(* Logix 5000 project; controller CarbonScout_MK6 vendor 1 type 14 code 154 rev 32.11; software revision 32.00; part 6 of 17 *)
(* tags used below, declared in another part *)
   Inp_OvrdCmd : DINT;   // Override Mode Command: 0=None, 1=Close, 2=Open
   Cfg_FailOpen : BOOL;   // 1=Fail Open (energize to close), 0=Fail Closed (energize to open)
   Cfg_PCmdClear : ALIAS FOR Mode.Cfg_PCmdClear;
   PSet_Owner : DINT;   // Program Owner Request ID (non-zero) or Release (zero)
   PCmd_Open : BOOL;   // Program Command to Open Valve
   PCmd_Close : BOOL;   // Program Command to Close Valve
   PCmd_Reset : BOOL;   // Program Command to Reset all Alarms requiring Reset
   OCmd_Open : BOOL;   // Operator Command to Open Valve
   OCmd_Close : BOOL;   // Operator Command to Close Valve
   OCmd_Bypass : BOOL;   // Operator Command to Bypass all Bypassable Interlocks and Permissives
   OCmd_Check : BOOL;   // Operator Command to Check (not bypass) all Interlocks and Permissives
   MCmd_Disable : BOOL;   // Maintenance Command to Disable Valve
   MCmd_Enable : BOOL;   // Maintenance Command to Enable (allow to energize) Valve
   OCmd_Reset : BOOL;   // Operator Command to Reset all Alarms requiring Reset
   OCmd_ResetAckAll : BOOL;   // Operator Command to Reset all Alarms and latched Shed conditions
   Out : BOOL;   // 1=Energize Valve Solenoid
   SrcQ_IO : DINT;   // Source and Quality of primary I/O (enumeration)
   SrcQ : DINT;   // Source and Quality of primary Val/Sts (enumeration)
   Val_Cmd : DINT;   // Device Command 0=None, 1=Close, 2=Open
   Val_Fdbk : DINT;   // Device Feedback 0=Moving, 1=Closed, 2=Opened, 3=Limit Switch Failure
   Val_Sts : DINT;   // Device Confirmed Sts 0=? 1=Closed 2=Open 5=Closing, 6=Opening, 33=Disabled
   Val_Fault : DINT;   // Device Fault Status 0=None, 16=Transit Stall, 17 = Full Stall, 32=I/O Fault, 34=Config Error
   Val_Mode : ALIAS FOR Mode.Val;
   Val_Owner : DINT;   // Current Object Owner ID (0=not owned)
   Val_Notify : DINT;   // Current Alarm Level and Acknowledgement (enumeration)
   Nrdy_Fail : BOOL;   // 1=Device Not Ready: Device Failure (Shed Requires Reset)
   Nrdy_IOFault : BOOL;   // 1=Device Not Ready: I/O Fault (Shed Requires Reset)
   Sts_MaintByp : BOOL;   // 1=A Maintenance Bypass is Active, display icon
   Sts_AlmInh : BOOL;   // 1=An Alarm is Shelved, Disabled or Suppressed, display icon
   Sts_Maint : ALIAS FOR Mode.Sts_Maint;
   Sts_Oper : ALIAS FOR Mode.Sts_Oper;
   Sts_NoMode : ALIAS FOR Mode.Sts_NoMode;
   Sts_IOFault : ALIAS FOR IOFault.Inp;   // I/O Comm Fault Status (0=OK, 1=Bad)
   Rdy_Disable : BOOL;   // 1=Ready to receive MCmd_Disable (enables HMI button)
   Rdy_Enable : BOOL;   // 1=Ready to receive MCmd_Enable (enables HMI button)
   Rdy_Reset : BOOL;   // 1=Ready to receive OCmd_Reset (enables HMI button)
   Rdy_ResetAckAll : BOOL;   // 1=At least one Alarm or latched Shed condition requires Reset or Ack
   P_ValveSO : BOOL;   // Unique Parameter Name for auto - discovery
   Mode : P_Mode;   // Valve Mode Selection
   IOFault : P_Alarm;   // I/O Fault Alarm
   IntlkTrip : P_Alarm;   // Interlock Trip Alarm
   TransitStall : P_Alarm;   // Valve Transit Stall (moved but did not reach target) Alarm
   FullStall : P_Alarm;   // Valve Full Stall (did not move) Alarm
   Wrk_Open : BOOL;   // 1=Requested to OPEN Valve, 0=Requested to CLOSE Valve
   Wrk_SimOpenT : TIMER;   // Simulation Delay until Opened
   Wrk_SimCloseT : TIMER;   // Simulation Delay until Closed
   Wrk_Notify : DINT;   // Buffer for building Val_Notify
   Wrk_TransitStallT : TIMER;   // Timer for Transit Stall Check
   Wrk_FullStallT : TIMER;   // Timer for Full Stall Check
   Wrk_SimOpenLS : BOOL;   // Simulated valve Open Limit Switch
   Wrk_SimClosedLS : BOOL;   // Simulated valve Closed Limit Switch
   test : DINT;
(* P_ValveSO, continued *)

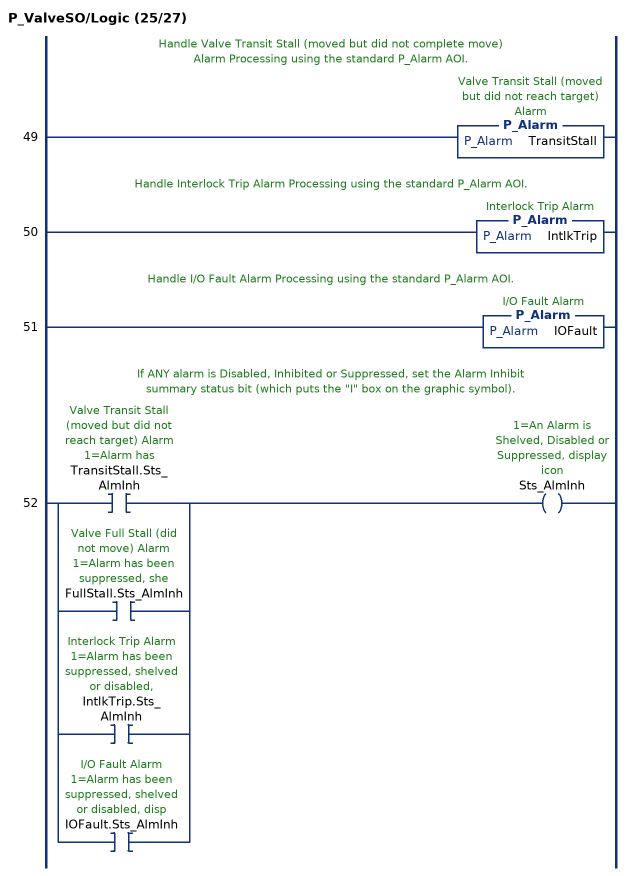
   // Handle Valve Transit Stall (moved but did not complete move)
   // Alarm Processing using the standard P_Alarm AOI.
   49: P_Alarm(TransitStall);
   // Handle Interlock Trip Alarm Processing using the standard P_Alarm AOI.
   50: P_Alarm(IntlkTrip);
   // Handle I/O Fault Alarm Processing using the standard P_Alarm AOI.
   51: P_Alarm(IOFault);
   // If ANY alarm is Disabled, Inhibited or Suppressed, set the Alarm Inhibit
   // summary status bit (which puts the "I" box on the graphic symbol).
   52: [XIC(TransitStall.Sts_AlmInh) ,XIC(FullStall.Sts_AlmInh) ,XIC(IntlkTrip.Sts_AlmInh) ,XIC(IOFault.Sts_AlmInh) ]OTE(Sts_AlmInh);
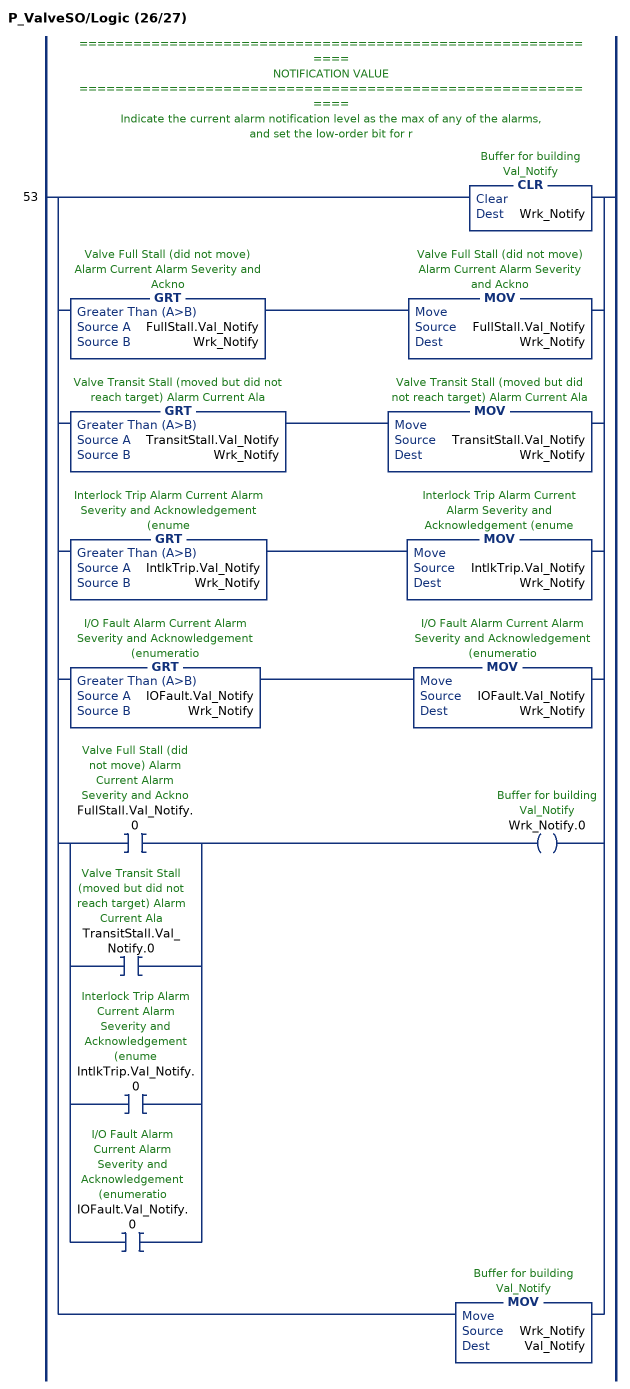
   // ============================================================
   // NOTIFICATION VALUE
   // ============================================================
   // Indicate the current alarm notification level as the max of any of the alarms,
   // and set the low-order bit for r
   53: [CLR(Wrk_Notify) ,GRT(FullStall.Val_Notify,Wrk_Notify) MOV(FullStall.Val_Notify,Wrk_Notify) ,GRT(TransitStall.Val_Notify,Wrk_Notify) MOV(TransitStall.Val_Notify,Wrk_Notify) ,GRT(IntlkTrip.Val_Notify,Wrk_Notify) MOV(IntlkTrip.Val_Notify,Wrk_Notify) ,GRT(IOFault.Val_Notify,Wrk_Notify) MOV(IOFault.Val_Notify,Wrk_Notify) ,[XIC(FullStall.Val_Notify.0) ,XIC(TransitStall.Val_Notify.0) ,XIC(IntlkTrip.Val_Notify.0) ,XIC(IOFault.Val_Notify.0) ] OTE(Wrk_Notify.0) ,MOV(Wrk_Notify,Val_Notify) ];
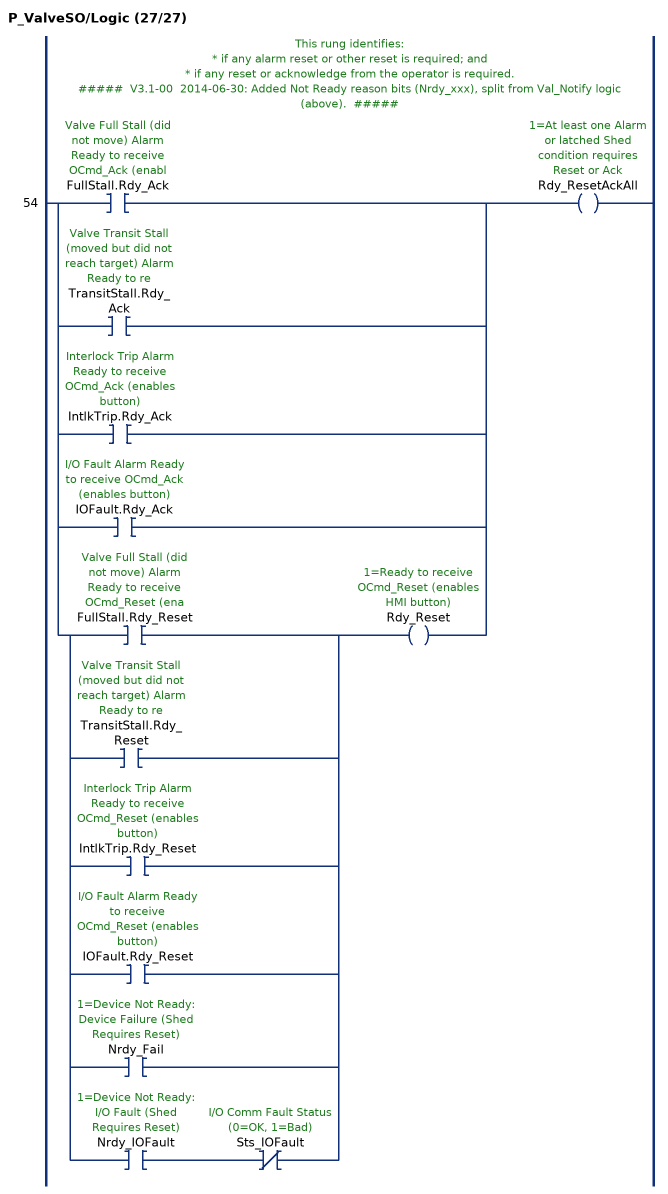
   // This rung identifies:
   // * if any alarm reset or other reset is required; and
   // * if any reset or acknowledge from the operator is required.
   // #####  V3.1-00  2014-06-30: Added Not Ready reason bits (Nrdy_xxx), split from Val_Notify logic (above).  #####
   54: [[XIC(FullStall.Rdy_Ack) ,XIC(TransitStall.Rdy_Ack) ,XIC(IntlkTrip.Rdy_Ack) ,XIC(IOFault.Rdy_Ack) ] ,[XIC(FullStall.Rdy_Reset) ,XIC(TransitStall.Rdy_Reset) ,XIC(IntlkTrip.Rdy_Reset) ,XIC(IOFault.Rdy_Reset) ,XIC(Nrdy_Fail) ,XIC(Nrdy_IOFault) XIO(Sts_IOFault) ] OTE(Rdy_Reset) ]OTE(Rdy_ResetAckAll);
END_ROUTINE

ROUTINE Prescan   (* ladder *)
// Clear Ownership, set to De-Energized state, clear "lurking" Commands
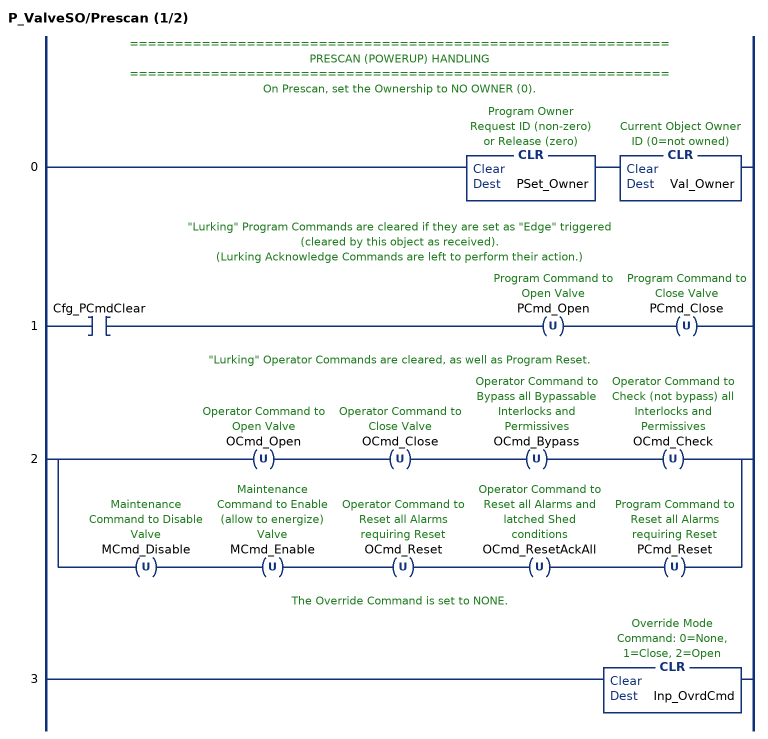
   // ============================================================
   // PRESCAN (POWERUP) HANDLING
   // ============================================================
   // On Prescan, set the Ownership to NO OWNER (0).
   0: CLR(PSet_Owner)CLR(Val_Owner);
   // "Lurking" Program Commands are cleared if they are set as "Edge" triggered
   // (cleared by this object as received).
   // (Lurking Acknowledge Commands are left to perform their action.)
   1: XIC(Cfg_PCmdClear)OTU(PCmd_Open)OTU(PCmd_Close);
   // "Lurking" Operator Commands are cleared, as well as Program Reset.
   2: [OTU(OCmd_Open) OTU(OCmd_Close) OTU(OCmd_Bypass) OTU(OCmd_Check) ,OTU(MCmd_Disable) OTU(MCmd_Enable) OTU(OCmd_Reset) OTU(OCmd_ResetAckAll) OTU(PCmd_Reset) ];
   // The Override Command is set to NONE.
   3: CLR(Inp_OvrdCmd);
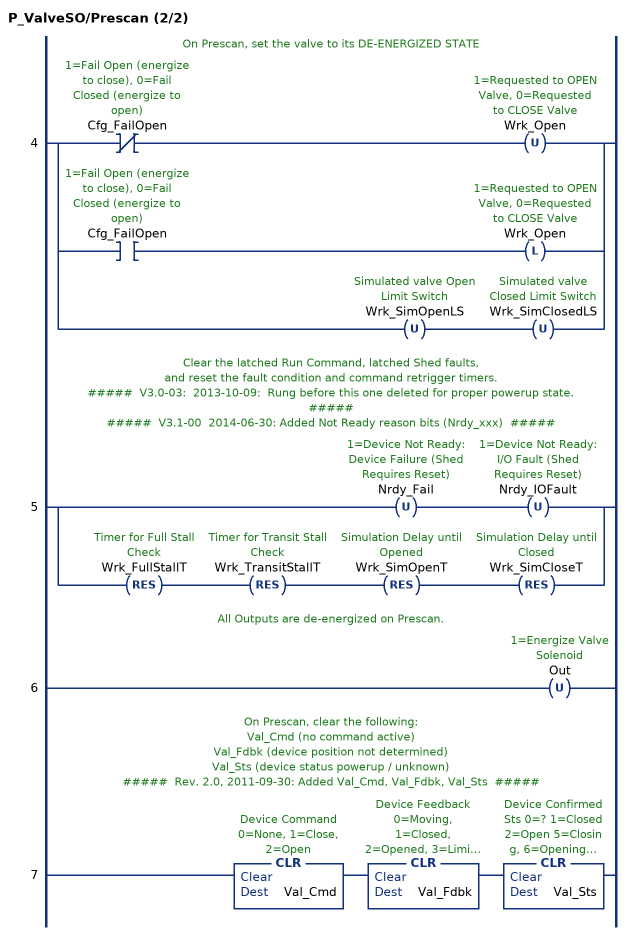
   // On Prescan, set the valve to its DE-ENERGIZED STATE
   4: [XIO(Cfg_FailOpen) OTU(Wrk_Open) ,XIC(Cfg_FailOpen) OTL(Wrk_Open) ,OTU(Wrk_SimOpenLS) OTU(Wrk_SimClosedLS) ];
   // Clear the latched Run Command, latched Shed faults,
   // and reset the fault condition and command retrigger timers.
   // #####  V3.0-03:  2013-10-09:  Rung before this one deleted for proper powerup state.  #####
   // #####  V3.1-00  2014-06-30: Added Not Ready reason bits (Nrdy_xxx)  #####
   5: [OTU(Nrdy_Fail) OTU(Nrdy_IOFault) ,RES(Wrk_FullStallT) RES(Wrk_TransitStallT) RES(Wrk_SimOpenT) RES(Wrk_SimCloseT) ];
   // All Outputs are de-energized on Prescan.
   6: OTU(Out);
   // On Prescan, clear the following:
   // Val_Cmd (no command active)
   // Val_Fdbk (device position not determined)
   // Val_Sts (device status powerup / unknown)
   // #####  Rev. 2.0, 2011-09-30: Added Val_Cmd, Val_Fdbk, Val_Sts  #####
   7: CLR(Val_Cmd)CLR(Val_Fdbk)CLR(Val_Sts);
END_ROUTINE
END_ADD_ON_INSTRUCTION

ADD_ON_INSTRUCTION TimerCompare   (* revision 1.0, ExecutePrescan *)
VAR_INPUT
   In_PresetTime1 : DINT; {required}
   In_PresetTime1_Multiplier : DINT; {required}
   In_PresetTime2 : DINT; {required}
   In_PresetTime2_Multiplier : DINT; {required}
   In_Time : DINT; {required}
END_VAR
VAR_OUTPUT
   Out_DN : BOOL;
END_VAR
VAR_INPUT
   In_ActiveStep : DINT; {required}
END_VAR
VAR
   Local_Time1 : DINT; {access None}
   Local_Time2 : DINT; {access None}
   Local_Time3 : DINT; {access None}
   LocalTimerDB : TIMER; {access None}
   LocalActiveStep : DINT; {access None}
END_VAR

ROUTINE Logic   (* ladder *)
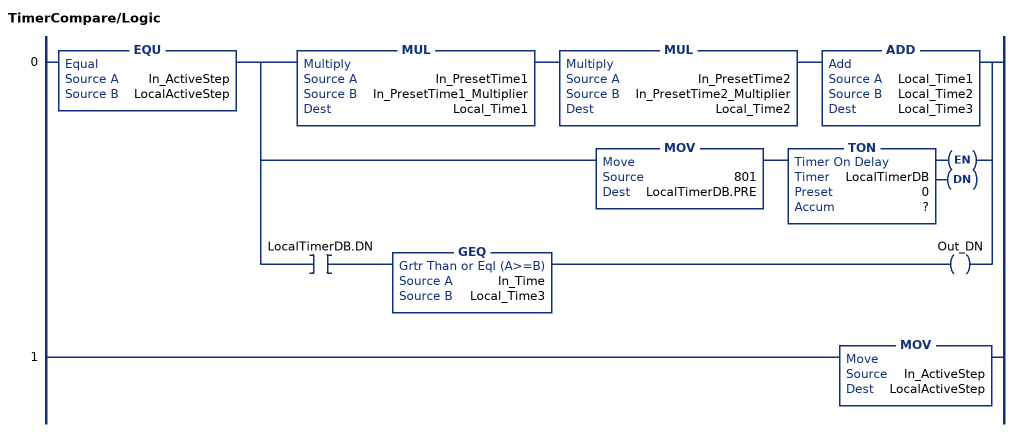
   0: EQU(In_ActiveStep,LocalActiveStep)[MUL(In_PresetTime1,In_PresetTime1_Multiplier,Local_Time1) MUL(In_PresetTime2,In_PresetTime2_Multiplier,Local_Time2) ADD(Local_Time1,Local_Time2,Local_Time3) ,MOV(801,LocalTimerDB.PRE) TON(LocalTimerDB,?,?) ,XIC(LocalTimerDB.DN) GEQ(In_Time,Local_Time3) OTE(Out_DN) ];
   1: MOV(In_ActiveStep,LocalActiveStep);
END_ROUTINE

ROUTINE Prescan   (* ladder *)
// Prescan
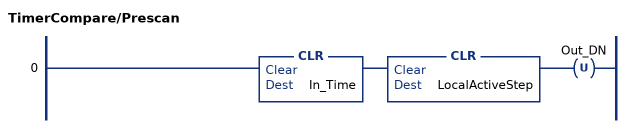
   0: CLR(In_Time)CLR(LocalActiveStep)OTU(Out_DN);
END_ROUTINE
END_ADD_ON_INSTRUCTION

ADD_ON_INSTRUCTION TimeRemainingCal   (* revision 1.0 *)
VAR_INPUT
   In_PresetTime : DINT; {visible}   // sec
END_VAR
VAR_OUTPUT
   RemainingHr : DINT; {required}
   RemainingMin : DINT; {required}
   RemainingSec : DINT; {required}
END_VAR
VAR_INPUT
   In_Time : DINT; {required}   // sec
END_VAR
VAR
   Local_Remaining : DINT; {access None}
   Local_RemainingMin : DINT; {access None}
   Local_Remainingsec : DINT; {access None}
END_VAR

ROUTINE Logic   (* ladder *)
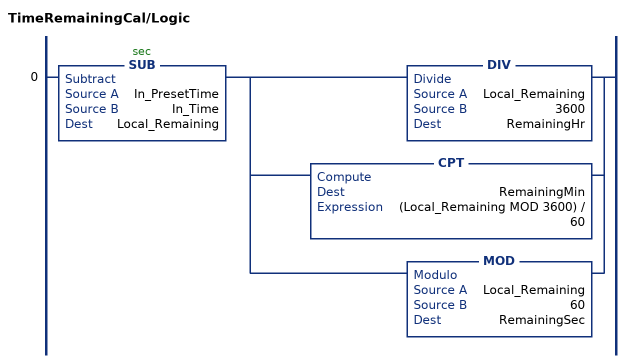
   0: SUB(In_PresetTime,In_Time,Local_Remaining)[DIV(Local_Remaining,3600,RemainingHr) ,CPT(RemainingMin,(Local_Remaining MOD 3600) / 60) ,MOD(Local_Remaining,60,RemainingSec) ];
END_ROUTINE
END_ADD_ON_INSTRUCTION

VAR_GLOBAL   (* controller tags *)
   a_Software_Version : STRING := '2.0.0';   // This must be updated and have a corrosponding change log and compadibility doc
   AI_AIT_01 : P_AIn := (Inp_PV := 9.085448, Inp_HiHiGate := 1, Inp_HiGate := 1, Inp_LoGate := 1, Inp_LoLoGate := 1, Inp_FailGate := 1, Cfg_SetTrack := 1, Cfg_PCmdClear := 1, Cfg_HiHiAckReqd := 1, Cfg_HiAckReqd := 1, Cfg_LoAckReqd := 1, Cfg_LoLoAckReqd := 1, Cfg_FailAckReqd := 1, Cfg_HiHiSeverity := 750, Cfg_HiSeverity := 500, Cfg_LoSeverity := 500, Cfg_LoLoSeverity := 750, Cfg_FailSeverity := 1000, Cfg_InpRawMax := 14.0, Cfg_PVEUMax := 14.0, Cfg_HiHiDB := 1.0, Cfg_HiDB := 1.0, Cfg_LoDB := 1.0, Cfg_LoLoDB := 1.0, Cfg_FailHiLim := 103.958336, Cfg_FailLoLim := -2.0833333, Cfg_FailDB := 0.41666666, Cfg_FailGateDly := 10, PSet_HiHiLim := 1.5e+38, PSet_HiLim := 1.5e+38, PSet_LoLim := -1.5e+38, PSet_LoLoLim := -1.5e+38, MSet_SubstPV := 9.085448, OSet_HiHiLim := 1.5e+38, OSet_HiLim := 1.5e+38, OSet_LoLim := -1.5e+38, OSet_LoLoLim := -1.5e+38, Set_SimPV := 9.085448, Val := 9.085448, Val_InpPV := 9.085448, Val_PVMinCapt := 9.085448, Val_PVMaxCapt := 9.085448, Val_PVEUMax := 14.0, SrcQ_IO := 1, SrcQ := 1, Val_Mode := 9, Val_HiHiLim := 1.5e+38, Val_HiLim := 1.5e+38, Val_LoLim := -1.5e+38, Val_LoLoLim := -1.5e+38, Sts_InpPV := 1, Sts_Oper := 1, Sts_HiHiGate := 1, Ack_HiHi := 1, Sts_HiGate := 1, Ack_Hi := 1, Sts_LoGate := 1, Ack_Lo := 1, Sts_LoLoGate := 1, Ack_LoLo := 1,
        Sts_FailGate := 1, Ack_Fail := 1, Rdy_OSet := 1);   // pH
   AI_AIT_02 : P_AIn := (Inp_PV := 6.017242, Inp_HiHiGate := 1, Inp_HiGate := 1, Inp_LoGate := 1, Inp_LoLoGate := 1, Inp_FailGate := 1, Cfg_SetTrack := 1, Cfg_PCmdClear := 1, Cfg_HiHiAckReqd := 1, Cfg_HiAckReqd := 1, Cfg_LoAckReqd := 1, Cfg_LoLoAckReqd := 1, Cfg_FailAckReqd := 1, Cfg_HiHiSeverity := 750, Cfg_HiSeverity := 500, Cfg_LoSeverity := 500, Cfg_LoLoSeverity := 750, Cfg_FailSeverity := 1000, Cfg_InpRawMax := 50.0, Cfg_PVEUMax := 50.0, Cfg_HiHiDB := 1.0, Cfg_HiDB := 1.0, Cfg_LoDB := 1.0, Cfg_LoLoDB := 1.0, Cfg_FailHiLim := 103.958336, Cfg_FailLoLim := -2.0833333, Cfg_FailDB := 0.41666666, Cfg_FailGateDly := 5, PSet_HiHiLim := 15000.0, PSet_HiLim := 15000.0, PSet_LoLim := -15000.0, PSet_LoLoLim := 15000.0, MSet_SubstPV := 39.0, OSet_HiHiLim := 15000.0, OSet_HiLim := 15000.0, OSet_LoLim := -15000.0, OSet_LoLoLim := 15000.0, Set_SimPV := 6.017242, Val := 39.0, Val_InpPV := 6.017242, Val_PVMinCapt := 39.0, Val_PVMaxCapt := 39.0, Val_PVEUMax := 50.0, SrcQ_IO := 1, SrcQ := 18, Val_Fault := 24, Val_Mode := 2, Val_HiHiLim := 15000.0, Val_HiLim := 15000.0, Val_LoLim := -15000.0, Val_LoLoLim := 15000.0, Sts_SubstPV := 1, Sts_MaintByp := 1, Sts_Maint := 1, Sts_HiHiGate := 1, Ack_HiHi := 1, Sts_HiGate := 1, Ack_Hi := 1, Sts_LoGate := 1, Ack_Lo := 1,
        Sts_LoLoCmp := 1, Sts_LoLoGate := 1, Sts_LoLo := 1, Ack_LoLo := 1, Sts_FailGate := 1, Ack_Fail := 1, Rdy_InpPV := 1, Rdy_OSet := 1);   // DO
   AI_AIT_03 : P_AIn := (Inp_HiHiGate := 1, Inp_HiGate := 1, Inp_LoGate := 1, Inp_LoLoGate := 1, Inp_FailGate := 1, Cfg_SetTrack := 1, Cfg_PCmdClear := 1, Cfg_HiHiAckReqd := 1, Cfg_HiAckReqd := 1, Cfg_LoAckReqd := 1, Cfg_LoLoAckReqd := 1, Cfg_FailAckReqd := 1, Cfg_HiHiSeverity := 750, Cfg_HiSeverity := 500, Cfg_LoSeverity := 500, Cfg_LoLoSeverity := 750, Cfg_FailSeverity := 1000, Cfg_InpRawMax := 100.0, Cfg_PVEUMax := 100.0, Cfg_HiHiDB := 1.0, Cfg_HiDB := 1.0, Cfg_LoDB := 1.0, Cfg_LoLoDB := 1.0, Cfg_FailHiLim := 103.958336, Cfg_FailLoLim := -2.0833333, Cfg_FailDB := 0.41666666, PSet_HiHiLim := 1.5e+38, PSet_HiLim := 1.5e+38, PSet_LoLim := -1.5e+38, PSet_LoLoLim := -1.5e+38, OSet_HiHiLim := 1.5e+38, OSet_HiLim := 1.5e+38, OSet_LoLim := -1.5e+38, OSet_LoLoLim := -1.5e+38, Val_PVMinCapt := 1.5e+38, Val_PVMaxCapt := -1.5e+38, Val_PVEUMax := 100.0, Val_HiHiLim := 1.5e+38, Val_HiLim := 1.5e+38, Val_LoLim := -1.5e+38, Val_LoLoLim := -1.5e+38, Sts_InpPV := 1, Sts_Oper := 1, Ack_HiHi := 1, Ack_Hi := 1, Ack_Lo := 1, Ack_LoLo := 1, Ack_Fail := 1);
   AI_Booster : P_AIn := (Inp_PV := 18408.0, Inp_HiHiGate := 1, Inp_HiGate := 1, Inp_LoGate := 1, Inp_LoLoGate := 1, Inp_FailGate := 1, Cfg_SetTrack := 1, Cfg_PCmdClear := 1, Cfg_HiHiAckReqd := 1, Cfg_HiAckReqd := 1, Cfg_LoAckReqd := 1, Cfg_LoLoAckReqd := 1, Cfg_FailAckReqd := 1, Cfg_HiHiSeverity := 750, Cfg_HiSeverity := 500, Cfg_LoSeverity := 500, Cfg_LoLoSeverity := 750, Cfg_FailSeverity := 1000, Cfg_InpRawMin := 4000.0, Cfg_InpRawMax := 20000.0, Cfg_PVEUMax := 100.0, Cfg_HiHiDB := 1.0, Cfg_HiDB := 1.0, Cfg_LoDB := 1.0, Cfg_LoOnDly := 1, Cfg_LoLoDB := 1.0, Cfg_LoLoOnDly := 1, Cfg_FailHiLim := 103.958336, Cfg_FailLoLim := -2.0833333, Cfg_FailDB := 0.41666666, PSet_HiHiLim := 95.0, PSet_HiLim := 80.0, PSet_LoLim := 25.0, PSet_LoLoLim := 10.0, MSet_SubstPV := 89.91875, OSet_HiHiLim := 95.0, OSet_HiLim := 80.0, OSet_LoLim := 25.0, OSet_LoLoLim := 10.0, Set_SimPV := 89.91875, Val := 89.91875, Val_InpPV := 89.91875, Val_PVMinCapt := 85.05625, Val_PVMaxCapt := 91.4, Val_PVEUMax := 100.0, SrcQ_IO := 1, SrcQ := 1, Val_Fault := 21, Val_Mode := 9, Val_HiHiLim := 95.0, Val_HiLim := 80.0, Val_LoLim := 25.0, Val_LoLoLim := 10.0, Sts_InpPV := 1, Sts_Oper := 1, Sts_HiHiGate := 1, Ack_HiHi := 1, Sts_HiCmp := 1, Sts_HiGate := 1, Sts_Hi := 1,
        Ack_Hi := 1, Sts_LoGate := 1, Ack_Lo := 1, Sts_LoLoGate := 1, Ack_LoLo := 1, Sts_FailGate := 1, Ack_Fail := 1, Rdy_OSet := 1);   // Booster Tank Level
   AI_FIT_01 : P_AIn := (Inp_PV := 4000.0, Inp_HiHiGate := 1, Inp_HiGate := 1, Inp_FailGate := 1, Cfg_SetTrack := 1, Cfg_PCmdClear := 1, Cfg_HasLoLoAlm := 1, Cfg_HasFailAlm := 1, Cfg_HiHiAckReqd := 1, Cfg_HiAckReqd := 1, Cfg_LoAckReqd := 1, Cfg_HiHiSeverity := 750, Cfg_HiSeverity := 500, Cfg_LoSeverity := 500, Cfg_LoLoSeverity := 750, Cfg_FailSeverity := 1000, Cfg_InpRawMin := 4000.0, Cfg_InpRawMax := 20000.0, Cfg_PVEUMax := 50.0, Cfg_HiHiDB := 1.0, Cfg_HiDB := 1.0, Cfg_LoDB := 1.0, Cfg_LoOnDly := 5, Cfg_LoGateDly := 5, Cfg_LoLoDB := 1.0, Cfg_LoLoOnDly := 5, Cfg_LoLoGateDly := 5, Cfg_FailHiLim := 55.0, Cfg_FailLoLim := -5.0, Cfg_FailDB := 0.41666666, PSet_HiHiLim := 1.5e+38, PSet_HiLim := 1.5e+38, PSet_LoLim := 0.5, PSet_LoLoLim := 0.3, OSet_HiHiLim := 1.5e+38, OSet_HiLim := 1.5e+38, OSet_LoLim := 0.5, OSet_LoLoLim := 0.3, Val_PVEUMax := 50.0, SrcQ_IO := 1, SrcQ := 1, Val_Mode := 9, Val_HiHiLim := 1.5e+38, Val_HiLim := 1.5e+38, Val_LoLim := 0.5, Val_LoLoLim := 0.3, Sts_InpPV := 1, Sts_Oper := 1, Sts_HiHiGate := 1, Ack_HiHi := 1, Sts_HiGate := 1, Ack_Hi := 1, Sts_LoCmp := 1, Ack_Lo := 1, Sts_LoLoCmp := 1, Ack_LoLo := 1, Sts_FailGate := 1, Ack_Fail := 1, Rdy_OSet := 1);   // Purge water flow
   AI_LIT_01 : P_AIn := (Inp_PV := 20489.0, Inp_HiHiGate := 1, Inp_HiGate := 1, Inp_LoGate := 1, Inp_LoLoGate := 1, Inp_FailGate := 1, Cfg_SetTrack := 1, Cfg_HasChanObj := 1, Cfg_PCmdClear := 1, Cfg_HiHiAckReqd := 1, Cfg_HiAckReqd := 1, Cfg_LoAckReqd := 1, Cfg_LoLoAckReqd := 1, Cfg_HiHiSeverity := 750, Cfg_HiSeverity := 500, Cfg_LoSeverity := 500, Cfg_LoLoSeverity := 750, Cfg_FailSeverity := 1000, Cfg_InpRawMin := 4000.0, Cfg_InpRawMax := 20000.0, Cfg_PVEUMin := 192.0, Cfg_PVEUMax := 1410.0, Cfg_FiltTC := 0.2, Cfg_HiHiDB := 1.0, Cfg_HiDB := 1.0, Cfg_LoDB := 1.0, Cfg_LoLoDB := 1.0, Cfg_FailHiLim := 1480.0, Cfg_FailLoLim := 180.0, Cfg_FailDB := 5.0, Cfg_FailGateDly := 10, PSet_HiHiLim := 1475.0, PSet_HiLim := 1.5e+38, PSet_LoLim := -1.5e+38, PSet_LoLoLim := 180.0, MSet_SubstPV := 1447.2251, OSet_HiHiLim := 1475.0, OSet_HiLim := 1.5e+38, OSet_LoLim := -1.5e+38, OSet_LoLoLim := 180.0, Set_SimPV := 1447.2251, Val := 1447.2251, Val_InpPV := 1447.2251, Val_PVMinCapt := 1447.2251, Val_PVMaxCapt := 1447.2251, Val_PVEUMin := 192.0, Val_PVEUMax := 1410.0, SrcQ_IO := 1, SrcQ := 1, Val_Mode := 9, Val_HiHiLim := 1475.0, Val_HiLim := 1.5e+38, Val_LoLim := -1.5e+38, Val_LoLoLim := 180.0, Sts_InpPV := 1, Sts_Oper := 1, Sts_HiHiGate := 1, Ack_HiHi := 1, Sts_HiGate := 1, Ack_Hi := 1,
        Sts_LoGate := 1, Ack_Lo := 1, Sts_LoLoGate := 1, Ack_LoLo := 1, Sts_FailGate := 1, Ack_Fail := 1, Rdy_OSet := 1);   // Carbon Scout Laser Level Transmitter
   AI_LIT_02 : P_AIn := (Inp_PV := 0.0015260963, Inp_HiHiGate := 1, Inp_HiGate := 1, Inp_LoGate := 1, Inp_LoLoGate := 1, Inp_FailGate := 1, Cfg_SetTrack := 1, Cfg_PCmdClear := 1, Cfg_HasFailAlm := 1, Cfg_HiHiAckReqd := 1, Cfg_HiAckReqd := 1, Cfg_LoAckReqd := 1, Cfg_LoLoAckReqd := 1, Cfg_HiHiSeverity := 750, Cfg_HiSeverity := 500, Cfg_LoSeverity := 500, Cfg_LoLoSeverity := 750, Cfg_FailSeverity := 1000, Cfg_InpRawMax := 20.0, Cfg_PVEUMax := 20.0, Cfg_HiHiDB := 1.0, Cfg_HiDB := 1.0, Cfg_LoDB := 1.0, Cfg_LoLoDB := 1.0, Cfg_FailHiLim := 25.0, Cfg_FailLoLim := -1.0, Cfg_FailDB := 0.5, Cfg_FailGateDly := 10, PSet_HiHiLim := 20.0, PSet_HiLim := 1.5e+38, PSet_LoLoLim := 3.8, MSet_SubstPV := 0.0015260963, OSet_HiHiLim := 20.0, OSet_HiLim := 1.5e+38, OSet_LoLoLim := 3.8, Set_SimPV := 0.0015260963, Val := 0.0015260963, Val_InpPV := 0.0015260963, Val_PVMinCapt := 0.0015260963, Val_PVMaxCapt := 0.0015260963, Val_PVEUMax := 20.0, SrcQ_IO := 1, SrcQ := 1, Val_Fault := 24, Val_Mode := 2, Val_HiHiLim := 20.0, Val_HiLim := 1.5e+38, Val_LoLoLim := 3.8, Sts_InpPV := 1, Sts_Maint := 1, Sts_HiHiGate := 1, Ack_HiHi := 1, Sts_HiGate := 1, Ack_Hi := 1, Sts_LoGate := 1, Ack_Lo := 1, Sts_LoLoCmp := 1, Sts_LoLoGate := 1, Sts_LoLo := 1, Ack_LoLo := 1,
        Sts_FailGate := 1, Ack_Fail := 1, Rdy_SubstPV := 1, Rdy_OSet := 1);   // Carbon Scout Cone Level Transmitter
   AI_PIT_01 : P_AIn := (Inp_PV := 12000.0, Inp_HiHiGate := 1, Inp_HiGate := 1, Inp_LoGate := 1, Inp_LoLoGate := 1, Inp_FailGate := 1, Cfg_SetTrack := 1, Cfg_PCmdClear := 1, Cfg_HasLoAlm := 1, Cfg_HasLoLoAlm := 1, Cfg_HasFailAlm := 1, Cfg_HiHiAckReqd := 1, Cfg_HiAckReqd := 1, Cfg_HiHiSeverity := 750, Cfg_HiSeverity := 500, Cfg_LoSeverity := 500, Cfg_LoLoSeverity := 750, Cfg_FailSeverity := 1000, Cfg_InpRawMin := 4000.0, Cfg_InpRawMax := 20000.0, Cfg_PVEUMax := 1000.0, Cfg_FiltTC := 1.0, Cfg_HiHiDB := 1.0, Cfg_HiDB := 1.0, Cfg_LoDB := 1.0, Cfg_LoOnDly := 5, Cfg_LoLoDB := 1.0, Cfg_LoLoOnDly := 60, Cfg_FailHiLim := 1100.0, Cfg_FailLoLim := -100.0, Cfg_FailDB := 0.41666666, Cfg_FailGateDly := 5, PSet_HiHiLim := 650.0, PSet_HiLim := 630.0, PSet_LoLim := 120.0, PSet_LoLoLim := 90.0, MSet_SubstPV := 500.0, OSet_HiHiLim := 650.0, OSet_HiLim := 630.0, OSet_LoLim := 120.0, OSet_LoLoLim := 90.0, Set_SimPV := 500.0, Val := 500.0, Val_InpPV := 500.0, Val_PVMinCapt := 500.0, Val_PVMaxCapt := 500.0, Val_PVEUMax := 1000.0, SrcQ_IO := 1, SrcQ := 1, Val_Mode := 9, Val_HiHiLim := 650.0, Val_HiLim := 630.0, Val_LoLim := 120.0, Val_LoLoLim := 90.0, Sts_InpPV := 1, Sts_Oper := 1, Sts_HiHiGate := 1, Ack_HiHi := 1, Sts_HiGate := 1, Ack_Hi := 1,
        Sts_LoGate := 1, Ack_Lo := 1, Sts_LoLoGate := 1, Ack_LoLo := 1, Sts_FailGate := 1, Ack_Fail := 1, Rdy_OSet := 1);   // Water supply pressure
   AI_TIT_01 : P_AIn := (Inp_HiHiGate := 1, Inp_HiGate := 1, Inp_LoGate := 1, Inp_LoLoGate := 1, Inp_FailGate := 1, Cfg_SetTrack := 1, Cfg_PCmdClear := 1, Cfg_HiHiAckReqd := 1, Cfg_HiAckReqd := 1, Cfg_LoAckReqd := 1, Cfg_LoLoAckReqd := 1, Cfg_FailAckReqd := 1, Cfg_HiHiSeverity := 750, Cfg_HiSeverity := 500, Cfg_LoSeverity := 500, Cfg_LoLoSeverity := 750, Cfg_FailSeverity := 1000, Cfg_InpRawMax := 50.0, Cfg_PVEUMax := 50.0, Cfg_HiHiDB := 1.0, Cfg_HiDB := 1.0, Cfg_LoDB := 1.0, Cfg_LoLoDB := 1.0, Cfg_FailHiLim := 103.958336, Cfg_FailLoLim := -2.0833333, Cfg_FailDB := 0.41666666, Cfg_FailGateDly := 5, PSet_HiHiLim := 1.5e+38, PSet_HiLim := 1.5e+38, PSet_LoLim := -1.5e+38, PSet_LoLoLim := -1.5e+38, OSet_HiHiLim := 1.5e+38, OSet_HiLim := 1.5e+38, OSet_LoLim := -1.5e+38, OSet_LoLoLim := -1.5e+38, Val_PVEUMax := 50.0, SrcQ_IO := 1, SrcQ := 1, Val_Mode := 9, Val_HiHiLim := 1.5e+38, Val_HiLim := 1.5e+38, Val_LoLim := -1.5e+38, Val_LoLoLim := -1.5e+38, Sts_InpPV := 1, Sts_Oper := 1, Sts_HiHiGate := 1, Ack_HiHi := 1, Sts_HiGate := 1, Ack_Hi := 1, Sts_LoGate := 1, Ack_Lo := 1, Sts_LoLoGate := 1, Ack_LoLo := 1, Sts_FailGate := 1, Ack_Fail := 1, Rdy_OSet := 1);   // Temperature
   AI_WIT_01 : P_AIn := (Inp_PV := -5.0, Inp_HiHiGate := 1, Inp_HiGate := 1, Inp_LoGate := 1, Inp_LoLoGate := 1, Inp_FailGate := 1, Cfg_SetTrack := 1, Cfg_PCmdClear := 1, Cfg_HasFailAlm := 1, Cfg_HiHiAckReqd := 1, Cfg_HiAckReqd := 1, Cfg_LoAckReqd := 1, Cfg_LoLoAckReqd := 1, Cfg_HiHiSeverity := 750, Cfg_HiSeverity := 500, Cfg_LoSeverity := 500, Cfg_LoLoSeverity := 750, Cfg_FailSeverity := 1000, Cfg_InpRawMin := 4000.0, Cfg_InpRawMax := 20000.0, Cfg_PVEUMin := 2.0, Cfg_PVEUMax := 52.0, Cfg_FiltTC := 1.0, Cfg_HiHiDB := 1.0, Cfg_HiDB := 1.0, Cfg_LoDB := 1.0, Cfg_LoLoDB := 1.0, Cfg_FailHiLim := 52.5, Cfg_FailLoLim := -5.0, Cfg_FailDB := 0.5, Cfg_FailGateDly := 5, PSet_HiHiLim := 1.5e+38, PSet_HiLim := 1.5e+38, PSet_LoLim := -1.5e+38, PSet_LoLoLim := -1.5e+38, MSet_SubstPV := -10.521875, OSet_HiHiLim := 1.5e+38, OSet_HiLim := 1.5e+38, OSet_LoLim := -1.5e+38, OSet_LoLoLim := -1.5e+38, Set_SimPV := -10.521875, PCmd_ClearCapt := 1, Val := -10.52187, Val_InpPV := -10.515625, Val_PVMinCapt := -10.52187, Val_PVMaxCapt := -10.51875, Val_PVEUMin := 2.0, Val_PVEUMax := 52.0, SrcQ_IO := 32, SrcQ := 19, Val_HiHiLim := 1.5e+38, Val_HiLim := 1.5e+38, Val_LoLim := -1.5e+38, Val_LoLoLim := -1.5e+38, Sts_PVBad := 1, Sts_AlmInh := 1, Sts_NoMode := 1, Ack_HiHi := 1, Ack_Hi := 1, Ack_Lo := 1,
        Ack_LoLo := 1, Ack_Fail := 1);   // Weight measure
   Client_to_Gekko : DINT[10] := ([0] := 64);
        [0].0   // Command Start Carbon Scout
        [0].1   // Command Pause Carbon Scout
        [0].15   // Take Tank Offline 16
        [0].16   // Take Tank Offline 1
        [0].17   // Take Tank Offline 2
        [0].18   // Take Tank Offline 3
        [0].19   // Take Tank Offline 4
        [0].2   // Command Shutdown Carbon Scout
        [0].20   // Take Tank Offline 5
        [0].21   // Take Tank Offline 6
        [0].22   // Take Tank Offline 7
        [0].23   // Take Tank Offline 8
        [0].24   // Take Tank Offline 9
        [0].25   // Take Tank Offline 10
        [0].26   // Take Tank Offline 11
        [0].27   // Take Tank Offline 12
        [0].28   // Take Tank Offline 13
        [0].29   // Take Tank Offline 14
        [0].3   // Command All Drives / Valves to Auto
        [0].30   // Take Tank Offline 15
        [0].4   // Command - Reset All Faults / Alarms
        [0].5   // Command Crash Stop Carbon Scout
        [0].6   // Indicate Newmont water supply is ok
        [0].7   // Tank HOld Request
        [0].8   // Enable Remote mode
        [0].9   // Remote Auto/Man Request 1 = Auto, 0 = Man
   CS_Alarms : P_Alarm[80] := ([0].Cfg_Exists := 1, [0].Cfg_AllowShelve := 1, [0].Cfg_AllowDisable := 1, [0].Cfg_PCmdClear := 1, [0].Cfg_Severity := 750, [0].Cfg_AlmMinOnT := 5, [0].Cfg_MaxShelfT := 480, [0].PCfg_AllowExist := 1, [0].Ack := 1, [0].Rdy_Shelve := 1, [0].Rdy_Disable := 1, [0].Rdy_Test := 1, [1].Cfg_Exists := 1, [1].Cfg_ResetReqd := 1, [1].Cfg_AllowShelve := 1, [1].Cfg_AllowDisable := 1, [1].Cfg_PCmdClear := 1, [1].Cfg_Severity := 750, [1].Cfg_AlmMinOnT := 5, [1].Cfg_MaxShelfT := 480, [1].PCfg_AllowExist := 1, [1].Ack := 1, [1].Rdy_Shelve := 1, [1].Rdy_Disable := 1, [1].Rdy_Test := 1, [2].Cfg_Exists := 1, [2].Cfg_AllowShelve := 1, [2].Cfg_AllowDisable := 1, [2].Cfg_PCmdClear := 1, [2].Cfg_Severity := 750, [2].Cfg_AlmMinOnT := 5, [2].Cfg_MaxShelfT := 480, [2].PCfg_AllowExist := 1, [2].Ack := 1, [2].Rdy_Shelve := 1, [2].Rdy_Disable := 1, [2].Rdy_Test := 1, [3].Cfg_Exists := 1, [3].Cfg_AllowShelve := 1, [3].Cfg_AllowDisable := 1, [3].Cfg_PCmdClear := 1, [3].Cfg_Severity := 750, [3].Cfg_AlmMinOnT := 5, [3].Cfg_MaxShelfT := 480, [3].PCfg_AllowExist := 1, [3].Ack := 1, [3].Rdy_Shelve := 1, [3].Rdy_Disable := 1, [3].Rdy_Test := 1, [4].Cfg_Exists := 1, [4].Cfg_AllowShelve := 1, [4].Cfg_AllowDisable := 1, [4].Cfg_PCmdClear := 1, [4].Cfg_Severity := 750, [4].Cfg_AlmMinOnT := 5, [4].Cfg_MaxShelfT := 480, [4].PCfg_AllowExist := 1, [4].Ack := 1, [4].Rdy_Shelve := 1, [4].Rdy_Disable := 1,
        [4].Rdy_Test := 1, [5].Cfg_Exists := 1, [5].Cfg_AllowShelve := 1, [5].Cfg_AllowDisable := 1, [5].Cfg_PCmdClear := 1, [5].Cfg_Severity := 750, [5].Cfg_AlmMinOnT := 5, [5].Cfg_MaxShelfT := 480, [5].PCfg_AllowExist := 1, [5].Ack := 1, [5].Rdy_Shelve := 1, [5].Rdy_Disable := 1, [5].Rdy_Test := 1, [6].Cfg_Exists := 1, [6].Cfg_AllowShelve := 1, [6].Cfg_AllowDisable := 1, [6].Cfg_PCmdClear := 1, [6].Cfg_Severity := 750, [6].Cfg_AlmMinOnT := 5, [6].Cfg_MaxShelfT := 480, [6].PCfg_AllowExist := 1, [6].Ack := 1, [6].Rdy_Shelve := 1, [6].Rdy_Disable := 1, [6].Rdy_Test := 1, [7].Cfg_Exists := 1, [7].Cfg_AllowShelve := 1, [7].Cfg_AllowDisable := 1, [7].Cfg_PCmdClear := 1, [7].Cfg_Severity := 750, [7].Cfg_AlmMinOnT := 5, [7].Cfg_MaxShelfT := 480, [7].PCfg_AllowExist := 1, [7].Ack := 1, [7].Rdy_Shelve := 1, [7].Rdy_Disable := 1, [7].Rdy_Test := 1, [8].Cfg_Exists := 1, [8].Cfg_AllowShelve := 1, [8].Cfg_AllowDisable := 1, [8].Cfg_PCmdClear := 1, [8].Cfg_Severity := 750, [8].Cfg_AlmMinOnT := 5, [8].Cfg_MaxShelfT := 480, [8].PCfg_AllowExist := 1, [8].Ack := 1, [8].Rdy_Shelve := 1, [8].Rdy_Disable := 1, [8].Rdy_Test := 1, [9].Cfg_Exists := 1, [9].Cfg_AllowShelve := 1, [9].Cfg_AllowDisable := 1, [9].Cfg_PCmdClear := 1, [9].Cfg_Severity := 750, [9].Cfg_AlmMinOnT := 5, [9].Cfg_MaxShelfT := 480, [9].PCfg_AllowExist := 1, [9].Ack := 1, [9].Rdy_Shelve := 1, [9].Rdy_Disable := 1,
        [9].Rdy_Test := 1, [10].Cfg_Exists := 1, [10].Cfg_AllowShelve := 1, [10].Cfg_AllowDisable := 1, [10].Cfg_PCmdClear := 1, [10].Cfg_Severity := 750, [10].Cfg_AlmMinOnT := 5, [10].Cfg_MaxShelfT := 480, [10].PCfg_AllowExist := 1, [10].Ack := 1, [10].Rdy_Shelve := 1, [10].Rdy_Disable := 1, [10].Rdy_Test := 1, [11].Cfg_Exists := 1, [11].Cfg_AllowShelve := 1, [11].Cfg_AllowDisable := 1, [11].Cfg_PCmdClear := 1, [11].Cfg_Severity := 750, [11].Cfg_AlmMinOnT := 5, [11].Cfg_MaxShelfT := 480, [11].PCfg_AllowExist := 1, [11].Ack := 1, [11].Rdy_Shelve := 1, [11].Rdy_Disable := 1, [11].Rdy_Test := 1, [12].Cfg_Exists := 1, [12].Cfg_AllowShelve := 1, [12].Cfg_AllowDisable := 1, [12].Cfg_PCmdClear := 1, [12].Cfg_Severity := 750, [12].Cfg_AlmMinOnT := 5, [12].Cfg_MaxShelfT := 480, [12].PCfg_AllowExist := 1, [12].Ack := 1, [12].Rdy_Shelve := 1, [12].Rdy_Disable := 1, [12].Rdy_Test := 1, [13].Cfg_Exists := 1, [13].Cfg_AllowShelve := 1, [13].Cfg_AllowDisable := 1, [13].Cfg_PCmdClear := 1, [13].Cfg_Severity := 750, [13].Cfg_AlmMinOnT := 5, [13].Cfg_MaxShelfT := 480, [13].PCfg_AllowExist := 1, [13].Ack := 1, [13].Rdy_Shelve := 1, [13].Rdy_Disable := 1, [13].Rdy_Test := 1, [14].Cfg_Exists := 1, [14].Cfg_ResetReqd := 1, [14].Cfg_AllowShelve := 1, [14].Cfg_AllowDisable := 1, [14].Cfg_PCmdClear := 1, [14].Cfg_Severity := 750, [14].Cfg_AlmMinOnT := 5, [14].Cfg_MaxShelfT := 480, [14].PCfg_AllowExist := 1, [14].Ack := 1, [14].Rdy_Shelve := 1,
        [14].Rdy_Disable := 1, [14].Rdy_Test := 1, [15].Cfg_Exists := 1, [15].Cfg_ResetReqd := 1, [15].Cfg_AllowShelve := 1, [15].Cfg_AllowDisable := 1, [15].Cfg_PCmdClear := 1, [15].Cfg_Severity := 750, [15].Cfg_AlmMinOnT := 5, [15].Cfg_MaxShelfT := 480, [15].PCfg_AllowExist := 1, [15].Ack := 1, [15].Rdy_Shelve := 1, [15].Rdy_Disable := 1, [15].Rdy_Test := 1, [16].Cfg_Exists := 1, [16].Cfg_ResetReqd := 1, [16].Cfg_AllowShelve := 1, [16].Cfg_AllowDisable := 1, [16].Cfg_PCmdClear := 1, [16].Cfg_Severity := 750, [16].Cfg_AlmMinOnT := 5, [16].Cfg_MaxShelfT := 480, [16].PCfg_AllowExist := 1, [16].Ack := 1, [16].Rdy_Shelve := 1, [16].Rdy_Disable := 1, [16].Rdy_Test := 1, [17].Cfg_Exists := 1, [17].Cfg_ResetReqd := 1, [17].Cfg_AllowShelve := 1, [17].Cfg_AllowDisable := 1, [17].Cfg_PCmdClear := 1, [17].Cfg_Severity := 750, [17].Cfg_AlmMinOnT := 5, [17].Cfg_MaxShelfT := 480, [17].PCfg_AllowExist := 1, [17].Ack := 1, [17].Rdy_Shelve := 1, [17].Rdy_Disable := 1, [17].Rdy_Test := 1, [18].Cfg_Exists := 1, [18].Cfg_ResetReqd := 1, [18].Cfg_AllowShelve := 1, [18].Cfg_AllowDisable := 1, [18].Cfg_PCmdClear := 1, [18].Cfg_Severity := 750, [18].Cfg_AlmMinOnT := 5, [18].Cfg_MaxShelfT := 480, [18].PCfg_AllowExist := 1, [18].Ack := 1, [18].Rdy_Shelve := 1, [18].Rdy_Disable := 1, [18].Rdy_Test := 1, [19].Cfg_Exists := 1, [19].Cfg_ResetReqd := 1, [19].Cfg_AllowShelve := 1, [19].Cfg_AllowDisable := 1, [19].Cfg_PCmdClear := 1, [19].Cfg_Severity := 750,
        [19].Cfg_AlmMinOnT := 5, [19].Cfg_MaxShelfT := 480, [19].PCfg_AllowExist := 1, [19].Ack := 1, [19].Rdy_Shelve := 1, [19].Rdy_Disable := 1, [19].Rdy_Test := 1, [20].Cfg_Exists := 1, [20].Cfg_ResetReqd := 1, [20].Cfg_AllowShelve := 1, [20].Cfg_AllowDisable := 1, [20].Cfg_PCmdClear := 1, [20].Cfg_Severity := 750, [20].Cfg_AlmMinOnT := 5, [20].Cfg_MaxShelfT := 480, [20].PCfg_AllowExist := 1, [20].Ack := 1, [20].Rdy_Shelve := 1, [20].Rdy_Disable := 1, [20].Rdy_Test := 1, [21].Cfg_Exists := 1, [21].Cfg_ResetReqd := 1, [21].Cfg_AllowShelve := 1, [21].Cfg_AllowDisable := 1, [21].Cfg_PCmdClear := 1, [21].Cfg_Severity := 750, [21].Cfg_AlmMinOnT := 5, [21].Cfg_MaxShelfT := 480, [21].PCfg_AllowExist := 1, [21].Ack := 1, [21].Rdy_Shelve := 1, [21].Rdy_Disable := 1, [21].Rdy_Test := 1, [22].Cfg_Exists := 1, [22].Cfg_ResetReqd := 1, [22].Cfg_AllowShelve := 1, [22].Cfg_AllowDisable := 1, [22].Cfg_PCmdClear := 1, [22].Cfg_Severity := 750, [22].Cfg_AlmMinOnT := 5, [22].Cfg_MaxShelfT := 480, [22].PCfg_AllowExist := 1, [22].Ack := 1, [22].Rdy_Shelve := 1, [22].Rdy_Disable := 1, [22].Rdy_Test := 1, [23].Cfg_Exists := 1, [23].Cfg_ResetReqd := 1, [23].Cfg_AllowShelve := 1, [23].Cfg_AllowDisable := 1, [23].Cfg_PCmdClear := 1, [23].Cfg_Severity := 750, [23].Cfg_AlmMinOnT := 5, [23].Cfg_MaxShelfT := 480, [23].PCfg_AllowExist := 1, [23].Ack := 1, [23].Rdy_Shelve := 1, [23].Rdy_Disable := 1, [23].Rdy_Test := 1, [24].Cfg_Exists := 1,
        [24].Cfg_ResetReqd := 1, [24].Cfg_AllowShelve := 1, [24].Cfg_AllowDisable := 1, [24].Cfg_PCmdClear := 1, [24].Cfg_Severity := 750, [24].Cfg_AlmMinOnT := 5, [24].Cfg_MaxShelfT := 480, [24].PCfg_AllowExist := 1, [24].Ack := 1, [24].Rdy_Shelve := 1, [24].Rdy_Disable := 1, [24].Rdy_Test := 1, [25].Cfg_Exists := 1, [25].Cfg_AllowShelve := 1, [25].Cfg_AllowDisable := 1, [25].Cfg_PCmdClear := 1, [25].Cfg_Severity := 750, [25].Cfg_AlmMinOnT := 5, [25].Cfg_MaxShelfT := 480, [25].PCfg_AllowExist := 1, [25].Ack := 1, [25].Rdy_Shelve := 1, [25].Rdy_Disable := 1, [25].Rdy_Test := 1, [26].Cfg_Exists := 1, [26].Cfg_AllowShelve := 1, [26].Cfg_AllowDisable := 1, [26].Cfg_PCmdClear := 1, [26].Cfg_Severity := 750, [26].Cfg_AlmMinOnT := 5, [26].Cfg_MaxShelfT := 480, [26].PCfg_AllowExist := 1, [26].Ack := 1, [26].Rdy_Shelve := 1, [26].Rdy_Disable := 1, [26].Rdy_Test := 1, [27].Cfg_Exists := 1, [27].Cfg_AllowShelve := 1, [27].Cfg_AllowDisable := 1, [27].Cfg_PCmdClear := 1, [27].Cfg_Severity := 750, [27].Cfg_AlmMinOnT := 5, [27].Cfg_MaxShelfT := 480, [27].PCfg_AllowExist := 1, [27].Ack := 1, [27].Rdy_Shelve := 1, [27].Rdy_Disable := 1, [27].Rdy_Test := 1, [28].Cfg_Exists := 1, [28].Cfg_AllowShelve := 1, [28].Cfg_AllowDisable := 1, [28].Cfg_PCmdClear := 1, [28].Cfg_Severity := 750, [28].Cfg_AlmMinOnT := 5, [28].Cfg_MaxShelfT := 480, [28].PCfg_AllowExist := 1, [28].Ack := 1, [28].Rdy_Shelve := 1, [28].Rdy_Disable := 1, [28].Rdy_Test := 1,
        [29].Cfg_Exists := 1, [29].Cfg_AllowShelve := 1, [29].Cfg_AllowDisable := 1, [29].Cfg_PCmdClear := 1, [29].Cfg_Severity := 750, [29].Cfg_AlmMinOnT := 5, [29].Cfg_MaxShelfT := 480, [29].PCfg_AllowExist := 1, [29].Ack := 1, [29].Rdy_Shelve := 1, [29].Rdy_Disable := 1, [29].Rdy_Test := 1, [30].Cfg_Exists := 1, [30].Cfg_AllowShelve := 1, [30].Cfg_AllowDisable := 1, [30].Cfg_PCmdClear := 1, [30].Cfg_Severity := 750, [30].Cfg_AlmMinOnT := 5, [30].Cfg_MaxShelfT := 480, [30].PCfg_AllowExist := 1, [30].Ack := 1, [30].Rdy_Shelve := 1, [30].Rdy_Disable := 1, [30].Rdy_Test := 1, [31].Cfg_Exists := 1, [31].Cfg_AllowShelve := 1, [31].Cfg_AllowDisable := 1, [31].Cfg_PCmdClear := 1, [31].Cfg_Severity := 750, [31].Cfg_AlmMinOnT := 5, [31].Cfg_MaxShelfT := 480, [31].PCfg_AllowExist := 1, [31].Ack := 1, [31].Rdy_Shelve := 1, [31].Rdy_Disable := 1, [31].Rdy_Test := 1, [32].Cfg_Exists := 1, [32].Cfg_AllowShelve := 1, [32].Cfg_AllowDisable := 1, [32].Cfg_PCmdClear := 1, [32].Cfg_Severity := 750, [32].Cfg_AlmMinOnT := 5, [32].Cfg_MaxShelfT := 480, [32].PCfg_AllowExist := 1, [32].Ack := 1, [32].Rdy_Shelve := 1, [32].Rdy_Disable := 1, [32].Rdy_Test := 1, [33].Cfg_Exists := 1, [33].Cfg_AllowShelve := 1, [33].Cfg_AllowDisable := 1, [33].Cfg_PCmdClear := 1, [33].Cfg_Severity := 750, [33].Cfg_AlmMinOnT := 5, [33].Cfg_MaxShelfT := 480, [33].PCfg_AllowExist := 1, [33].Ack := 1, [33].Rdy_Shelve := 1, [33].Rdy_Disable := 1, [33].Rdy_Test := 1,
        [34].Cfg_Exists := 1, [34].Cfg_AllowShelve := 1, [34].Cfg_AllowDisable := 1, [34].Cfg_PCmdClear := 1, [34].Cfg_Severity := 750, [34].Cfg_AlmMinOnT := 5, [34].Cfg_MaxShelfT := 480, [34].PCfg_AllowExist := 1, [34].Ack := 1, [34].Rdy_Shelve := 1, [34].Rdy_Disable := 1, [34].Rdy_Test := 1, [35].Cfg_Exists := 1, [35].Cfg_AllowShelve := 1, [35].Cfg_AllowDisable := 1, [35].Cfg_PCmdClear := 1, [35].Cfg_Severity := 750, [35].Cfg_AlmMinOnT := 5, [35].Cfg_MaxShelfT := 480, [35].PCfg_AllowExist := 1, [35].Ack := 1, [35].Rdy_Shelve := 1, [35].Rdy_Disable := 1, [35].Rdy_Test := 1, [36].Cfg_Exists := 1, [36].Cfg_AllowShelve := 1, [36].Cfg_AllowDisable := 1, [36].Cfg_PCmdClear := 1, [36].Cfg_Severity := 750, [36].Cfg_AlmMinOnT := 5, [36].Cfg_MaxShelfT := 480, [36].PCfg_AllowExist := 1, [36].Ack := 1, [36].Rdy_Shelve := 1, [36].Rdy_Disable := 1, [36].Rdy_Test := 1, [37].Cfg_Exists := 1, [37].Cfg_AllowShelve := 1, [37].Cfg_AllowDisable := 1, [37].Cfg_PCmdClear := 1, [37].Cfg_Severity := 750, [37].Cfg_AlmMinOnT := 5, [37].Cfg_MaxShelfT := 480, [37].PCfg_AllowExist := 1, [37].Ack := 1, [37].Rdy_Shelve := 1, [37].Rdy_Disable := 1, [37].Rdy_Test := 1, [38].Cfg_Exists := 1, [38].Cfg_AllowShelve := 1, [38].Cfg_AllowDisable := 1, [38].Cfg_PCmdClear := 1, [38].Cfg_Severity := 750, [38].Cfg_AlmMinOnT := 5, [38].Cfg_MaxShelfT := 480, [38].PCfg_AllowExist := 1, [38].Ack := 1, [38].Rdy_Shelve := 1, [38].Rdy_Disable := 1, [38].Rdy_Test := 1,
        [39].Cfg_Exists := 1, [39].Cfg_AllowShelve := 1, [39].Cfg_AllowDisable := 1, [39].Cfg_PCmdClear := 1, [39].Cfg_Severity := 750, [39].Cfg_AlmMinOnT := 5, [39].Cfg_MaxShelfT := 480, [39].PCfg_AllowExist := 1, [39].Ack := 1, [39].Rdy_Shelve := 1, [39].Rdy_Disable := 1, [39].Rdy_Test := 1, [40].Cfg_Exists := 1, [40].Cfg_AllowShelve := 1, [40].Cfg_AllowDisable := 1, [40].Cfg_PCmdClear := 1, [40].Cfg_Severity := 750, [40].Cfg_AlmMinOnT := 5, [40].Cfg_MaxShelfT := 480, [40].PCfg_AllowExist := 1, [40].Ack := 1, [40].Rdy_Shelve := 1, [40].Rdy_Disable := 1, [40].Rdy_Test := 1, [41].Cfg_Exists := 1, [41].Cfg_AllowShelve := 1, [41].Cfg_AllowDisable := 1, [41].Cfg_PCmdClear := 1, [41].Cfg_Severity := 750, [41].Cfg_AlmMinOnT := 5, [41].Cfg_MaxShelfT := 480, [41].PCfg_AllowExist := 1, [41].Ack := 1, [41].Rdy_Shelve := 1, [41].Rdy_Disable := 1, [41].Rdy_Test := 1, [42].Inp := 1, [42].Cfg_Exists := 1, [42].Cfg_AllowShelve := 1, [42].Cfg_AllowDisable := 1, [42].Cfg_PCmdClear := 1, [42].Cfg_Severity := 750, [42].Cfg_AlmMinOnT := 5, [42].Cfg_MaxShelfT := 480, [42].PCfg_AllowExist := 1, [42].Val_Notify := 6, [42].Alm := 1, [42].Ack := 1, [42].Rdy_Shelve := 1, [42].Rdy_Disable := 1, [43].Inp := 1, [43].Cfg_Exists := 1, [43].Cfg_AllowShelve := 1, [43].Cfg_AllowDisable := 1, [43].Cfg_PCmdClear := 1, [43].Cfg_Severity := 750, [43].Cfg_AlmMinOnT := 5, [43].Cfg_MaxShelfT := 480, [43].PCfg_AllowExist := 1, [43].Val_Notify := 6,
        [43].Alm := 1, [43].Ack := 1, [43].Rdy_Shelve := 1, [43].Rdy_Disable := 1, [44].Cfg_Exists := 1, [44].Cfg_AllowShelve := 1, [44].Cfg_AllowDisable := 1, [44].Cfg_PCmdClear := 1, [44].Cfg_Severity := 736, [44].Cfg_AlmMinOnT := 5, [44].Cfg_MaxShelfT := 480, [44].PCfg_AllowExist := 1, [44].Ack := 1, [44].Rdy_Shelve := 1, [44].Rdy_Disable := 1, [44].Rdy_Test := 1, [45].Cfg_Exists := 1, [45].Cfg_AllowShelve := 1, [45].Cfg_AllowDisable := 1, [45].Cfg_PCmdClear := 1, [45].Cfg_Severity := 750, [45].Cfg_AlmMinOnT := 5, [45].Cfg_MaxShelfT := 480, [45].PCfg_AllowExist := 1, [45].Ack := 1, [45].Rdy_Shelve := 1, [45].Rdy_Disable := 1, [45].Rdy_Test := 1, [46].Cfg_Exists := 1, [46].Cfg_AllowShelve := 1, [46].Cfg_AllowDisable := 1, [46].Cfg_PCmdClear := 1, [46].Cfg_Severity := 750, [46].Cfg_AlmMinOnT := 5, [46].Cfg_MaxShelfT := 480, [46].PCfg_AllowExist := 1, [46].Ack := 1, [46].Rdy_Shelve := 1, [46].Rdy_Disable := 1, [46].Rdy_Test := 1, [47].Cfg_Exists := 1, [47].Cfg_AllowShelve := 1, [47].Cfg_AllowDisable := 1, [47].Cfg_PCmdClear := 1, [47].Cfg_Severity := 750, [47].Cfg_AlmMinOnT := 5, [47].Cfg_MaxShelfT := 480, [47].PCfg_AllowExist := 1, [47].Ack := 1, [47].Rdy_Shelve := 1, [47].Rdy_Disable := 1, [47].Rdy_Test := 1, [48].Cfg_Exists := 1, [48].Cfg_AllowShelve := 1, [48].Cfg_AllowDisable := 1, [48].Cfg_PCmdClear := 1, [48].Cfg_Severity := 750, [48].Cfg_AlmMinOnT := 5, [48].Cfg_MaxShelfT := 480, [48].PCfg_AllowExist := 1,
        [48].Ack := 1, [48].Rdy_Shelve := 1, [48].Rdy_Disable := 1, [48].Rdy_Test := 1, [49].Cfg_Exists := 1, [49].Cfg_AllowShelve := 1, [49].Cfg_AllowDisable := 1, [49].Cfg_PCmdClear := 1, [49].Cfg_Severity := 750, [49].Cfg_AlmMinOnT := 5, [49].Cfg_MaxShelfT := 480, [49].PCfg_AllowExist := 1, [49].Ack := 1, [49].Rdy_Shelve := 1, [49].Rdy_Disable := 1, [49].Rdy_Test := 1, [50].Cfg_Exists := 1, [50].Cfg_AllowShelve := 1, [50].Cfg_AllowDisable := 1, [50].Cfg_PCmdClear := 1, [50].Cfg_Severity := 750, [50].Cfg_AlmMinOnT := 5, [50].Cfg_MaxShelfT := 480, [50].PCfg_AllowExist := 1, [50].Ack := 1, [50].Rdy_Shelve := 1, [50].Rdy_Disable := 1, [50].Rdy_Test := 1, [51].Cfg_Exists := 1, [51].Cfg_AllowShelve := 1, [51].Cfg_AllowDisable := 1, [51].Cfg_PCmdClear := 1, [51].Cfg_Severity := 750, [51].Cfg_AlmMinOnT := 5, [51].Cfg_MaxShelfT := 480, [51].PCfg_AllowExist := 1, [51].Ack := 1, [51].Rdy_Shelve := 1, [51].Rdy_Disable := 1, [51].Rdy_Test := 1, [52].Cfg_Exists := 1, [52].Cfg_AllowShelve := 1, [52].Cfg_AllowDisable := 1, [52].Cfg_PCmdClear := 1, [52].Cfg_Severity := 750, [52].Cfg_AlmMinOnT := 5, [52].Cfg_MaxShelfT := 480, [52].PCfg_AllowExist := 1, [52].Ack := 1, [52].Rdy_Shelve := 1, [52].Rdy_Disable := 1, [52].Rdy_Test := 1, [53].Cfg_Exists := 1, [53].Cfg_AllowShelve := 1, [53].Cfg_AllowDisable := 1, [53].Cfg_PCmdClear := 1, [53].Cfg_Severity := 750, [53].Cfg_AlmMinOnT := 5, [53].Cfg_MaxShelfT := 480, [53].PCfg_AllowExist := 1,
        [53].Ack := 1, [53].Rdy_Shelve := 1, [53].Rdy_Disable := 1, [53].Rdy_Test := 1, [54].Cfg_Exists := 1, [54].Cfg_AllowShelve := 1, [54].Cfg_AllowDisable := 1, [54].Cfg_PCmdClear := 1, [54].Cfg_Severity := 750, [54].Cfg_AlmMinOnT := 5, [54].Cfg_MaxShelfT := 480, [54].PCfg_AllowExist := 1, [54].Ack := 1, [54].Rdy_Shelve := 1, [54].Rdy_Disable := 1, [54].Rdy_Test := 1, [55].Cfg_Exists := 1, [55].Cfg_AllowShelve := 1, [55].Cfg_AllowDisable := 1, [55].Cfg_PCmdClear := 1, [55].Cfg_Severity := 750, [55].Cfg_AlmMinOnT := 5, [55].Cfg_MaxShelfT := 480, [55].PCfg_AllowExist := 1, [55].Ack := 1, [55].Rdy_Shelve := 1, [55].Rdy_Disable := 1, [55].Rdy_Test := 1, [56].Cfg_Exists := 1, [56].Cfg_AllowShelve := 1, [56].Cfg_AllowDisable := 1, [56].Cfg_PCmdClear := 1, [56].Cfg_Severity := 750, [56].Cfg_AlmMinOnT := 5, [56].Cfg_MaxShelfT := 480, [56].PCfg_AllowExist := 1, [56].Ack := 1, [56].Rdy_Shelve := 1, [56].Rdy_Disable := 1, [56].Rdy_Test := 1, [57].Cfg_Exists := 1, [57].Cfg_ResetReqd := 1, [57].Cfg_AllowShelve := 1, [57].Cfg_AllowDisable := 1, [57].Cfg_PCmdClear := 1, [57].Cfg_Severity := 750, [57].Cfg_AlmMinOnT := 5, [57].Cfg_MaxShelfT := 480, [57].PCfg_AllowExist := 1, [57].Ack := 1, [57].Rdy_Shelve := 1, [57].Rdy_Disable := 1, [57].Rdy_Test := 1, [58].Cfg_Exists := 1, [58].Cfg_ResetReqd := 1, [58].Cfg_AllowShelve := 1, [58].Cfg_AllowDisable := 1, [58].Cfg_PCmdClear := 1, [58].Cfg_Severity := 750, [58].Cfg_AlmMinOnT := 5,
        [58].Cfg_MaxShelfT := 480, [58].PCfg_AllowExist := 1, [58].Ack := 1, [58].Rdy_Shelve := 1, [58].Rdy_Disable := 1, [58].Rdy_Test := 1, [59].Cfg_Exists := 1, [59].Cfg_ResetReqd := 1, [59].Cfg_AllowShelve := 1, [59].Cfg_AllowDisable := 1, [59].Cfg_PCmdClear := 1, [59].Cfg_Severity := 750, [59].Cfg_AlmMinOnT := 5, [59].Cfg_MaxShelfT := 480, [59].PCfg_AllowExist := 1, [59].Ack := 1, [59].Rdy_Shelve := 1, [59].Rdy_Disable := 1, [59].Rdy_Test := 1, [60].Cfg_Exists := 1, [60].Cfg_ResetReqd := 1, [60].Cfg_AllowShelve := 1, [60].Cfg_AllowDisable := 1, [60].Cfg_PCmdClear := 1, [60].Cfg_Severity := 750, [60].Cfg_AlmMinOnT := 5, [60].Cfg_MaxShelfT := 480, [60].PCfg_AllowExist := 1, [60].Ack := 1, [60].Rdy_Shelve := 1, [60].Rdy_Disable := 1, [60].Rdy_Test := 1, [61].Cfg_Exists := 1, [61].Cfg_ResetReqd := 1, [61].Cfg_AllowShelve := 1, [61].Cfg_AllowDisable := 1, [61].Cfg_PCmdClear := 1, [61].Cfg_Severity := 750, [61].Cfg_AlmMinOnT := 5, [61].Cfg_MaxShelfT := 480, [61].PCfg_AllowExist := 1, [61].Ack := 1, [61].Rdy_Shelve := 1, [61].Rdy_Disable := 1, [61].Rdy_Test := 1, [62].Cfg_Exists := 1, [62].Cfg_ResetReqd := 1, [62].Cfg_AllowShelve := 1, [62].Cfg_AllowDisable := 1, [62].Cfg_PCmdClear := 1, [62].Cfg_Severity := 750, [62].Cfg_AlmMinOnT := 5, [62].Cfg_MaxShelfT := 480, [62].PCfg_AllowExist := 1, [62].Ack := 1, [62].Rdy_Shelve := 1, [62].Rdy_Disable := 1, [62].Rdy_Test := 1, [63].Cfg_Exists := 1, [63].Cfg_AllowShelve := 1,
        [63].Cfg_AllowDisable := 1, [63].Cfg_PCmdClear := 1, [63].Cfg_Severity := 750, [63].Cfg_AlmMinOnT := 5, [63].Cfg_MaxShelfT := 480, [63].PCfg_AllowExist := 1, [63].Ack := 1, [63].Rdy_Shelve := 1, [63].Rdy_Disable := 1, [63].Rdy_Test := 1, [64].Cfg_Exists := 1, [64].Cfg_AllowShelve := 1, [64].Cfg_AllowDisable := 1, [64].Cfg_PCmdClear := 1, [64].Cfg_Severity := 750, [64].Cfg_AlmMinOnT := 5, [64].Cfg_MaxShelfT := 480, [64].PCfg_AllowExist := 1, [64].Ack := 1, [64].Rdy_Shelve := 1, [64].Rdy_Disable := 1, [64].Rdy_Test := 1, [65].Cfg_Exists := 1, [65].Cfg_AllowShelve := 1, [65].Cfg_AllowDisable := 1, [65].Cfg_PCmdClear := 1, [65].Cfg_Severity := 750, [65].Cfg_AlmMinOnT := 5, [65].Cfg_MaxShelfT := 480, [65].PCfg_AllowExist := 1, [65].Ack := 1, [65].Rdy_Shelve := 1, [65].Rdy_Disable := 1, [65].Rdy_Test := 1, [66].Cfg_Exists := 1, [66].Cfg_AllowShelve := 1, [66].Cfg_AllowDisable := 1, [66].Cfg_PCmdClear := 1, [66].Cfg_Severity := 750, [66].Cfg_AlmMinOnT := 5, [66].Cfg_MaxShelfT := 480, [66].PCfg_AllowExist := 1, [66].Ack := 1, [66].Rdy_Shelve := 1, [66].Rdy_Disable := 1, [66].Rdy_Test := 1, [67].Cfg_Exists := 1, [67].Cfg_AllowShelve := 1, [67].Cfg_AllowDisable := 1, [67].Cfg_PCmdClear := 1, [67].Cfg_Severity := 750, [67].Cfg_AlmMinOnT := 5, [67].Cfg_MaxShelfT := 480, [67].PCfg_AllowExist := 1, [67].Ack := 1, [67].Rdy_Shelve := 1, [67].Rdy_Disable := 1, [67].Rdy_Test := 1, [68].Cfg_Exists := 1, [68].Cfg_AllowShelve := 1,
        [68].Cfg_AllowDisable := 1, [68].Cfg_PCmdClear := 1, [68].Cfg_Severity := 750, [68].Cfg_AlmMinOnT := 5, [68].Cfg_MaxShelfT := 480, [68].PCfg_AllowExist := 1, [68].Ack := 1, [68].Rdy_Shelve := 1, [68].Rdy_Disable := 1, [68].Rdy_Test := 1, [69].Cfg_Exists := 1, [69].Cfg_AllowShelve := 1, [69].Cfg_AllowDisable := 1, [69].Cfg_PCmdClear := 1, [69].Cfg_Severity := 750, [69].Cfg_AlmMinOnT := 5, [69].Cfg_MaxShelfT := 480, [69].PCfg_AllowExist := 1, [69].Ack := 1, [69].Rdy_Shelve := 1, [69].Rdy_Disable := 1, [69].Rdy_Test := 1, [70].Cfg_Exists := 1, [70].Cfg_AllowShelve := 1, [70].Cfg_AllowDisable := 1, [70].Cfg_PCmdClear := 1, [70].Cfg_Severity := 750, [70].Cfg_AlmMinOnT := 5, [70].Cfg_MaxShelfT := 480, [70].PCfg_AllowExist := 1, [70].Ack := 1, [70].Disabled := 1, [70].Sts_AlmInh := 1, [70].Rdy_Shelve := 1, [70].Rdy_Enable := 1, [70].Rdy_Test := 1, [71].Cfg_Exists := 1, [71].Cfg_AllowShelve := 1, [71].Cfg_AllowDisable := 1, [71].Cfg_PCmdClear := 1, [71].Cfg_Severity := 750, [71].Cfg_AlmMinOnT := 5, [71].Cfg_MaxShelfT := 480, [71].PCfg_AllowExist := 1, [71].Ack := 1, [71].Disabled := 1, [71].Sts_AlmInh := 1, [71].Rdy_Shelve := 1, [71].Rdy_Enable := 1, [71].Rdy_Test := 1, [72].Cfg_Exists := 1, [72].Cfg_AllowShelve := 1, [72].Cfg_AllowDisable := 1, [72].Cfg_PCmdClear := 1, [72].Cfg_Severity := 750, [72].Cfg_AlmMinOnT := 5, [72].Cfg_MaxShelfT := 480, [72].PCfg_AllowExist := 1, [72].Ack := 1, [72].Rdy_Shelve := 1,
        [72].Rdy_Disable := 1, [72].Rdy_Test := 1, [73].Cfg_Exists := 1, [73].Cfg_AllowShelve := 1, [73].Cfg_AllowDisable := 1, [73].Cfg_PCmdClear := 1, [73].Cfg_Severity := 750, [73].Cfg_AlmMinOnT := 5, [73].Cfg_MaxShelfT := 480, [73].PCfg_AllowExist := 1, [73].Ack := 1, [73].Rdy_Shelve := 1, [73].Rdy_Disable := 1, [73].Rdy_Test := 1, [74].Cfg_Exists := 1, [74].Cfg_AllowShelve := 1, [74].Cfg_AllowDisable := 1, [74].Cfg_PCmdClear := 1, [74].Cfg_Severity := 750, [74].Cfg_AlmMinOnT := 5, [74].Cfg_MaxShelfT := 480, [74].PCfg_AllowExist := 1, [74].Ack := 1, [74].Rdy_Shelve := 1, [74].Rdy_Disable := 1, [74].Rdy_Test := 1, [75].Cfg_Exists := 1, [75].Cfg_AllowShelve := 1, [75].Cfg_AllowDisable := 1, [75].Cfg_PCmdClear := 1, [75].Cfg_Severity := 750, [75].Cfg_AlmMinOnT := 5, [75].Cfg_MaxShelfT := 480, [75].PCfg_AllowExist := 1, [75].Ack := 1, [75].Rdy_Shelve := 1, [75].Rdy_Disable := 1, [75].Rdy_Test := 1, [76].Cfg_Exists := 1, [76].Cfg_AllowShelve := 1, [76].Cfg_AllowDisable := 1, [76].Cfg_PCmdClear := 1, [76].Cfg_Severity := 750, [76].Cfg_AlmMinOnT := 5, [76].Cfg_MaxShelfT := 480, [76].PCfg_AllowExist := 1, [76].Ack := 1, [76].Rdy_Shelve := 1, [76].Rdy_Disable := 1, [76].Rdy_Test := 1, [77].Cfg_Exists := 1, [77].Cfg_AllowShelve := 1, [77].Cfg_AllowDisable := 1, [77].Cfg_PCmdClear := 1, [77].Cfg_Severity := 750, [77].Cfg_AlmMinOnT := 5, [77].Cfg_MaxShelfT := 480, [77].PCfg_AllowExist := 1, [77].Ack := 1, [77].Rdy_Shelve := 1,
        [77].Rdy_Disable := 1, [77].Rdy_Test := 1, [78].Cfg_Exists := 1, [78].Cfg_AllowShelve := 1, [78].Cfg_AllowDisable := 1, [78].Cfg_PCmdClear := 1, [78].Cfg_Severity := 750, [78].Cfg_AlmMinOnT := 5, [78].Cfg_MaxShelfT := 480, [78].PCfg_AllowExist := 1, [78].Ack := 1, [78].Rdy_Shelve := 1, [78].Rdy_Disable := 1, [78].Rdy_Test := 1, [79].Cfg_Exists := 1, [79].Cfg_AllowShelve := 1, [79].Cfg_AllowDisable := 1, [79].Cfg_PCmdClear := 1, [79].Cfg_Severity := 750, [79].Cfg_AlmMinOnT := 5, [79].Cfg_MaxShelfT := 480, [79].PCfg_AllowExist := 1, [79].Ack := 1, [79].Rdy_Shelve := 1, [79].Rdy_Disable := 1, [79].Rdy_Test := 1);
        [39]   // XRF Exposure Lasted Longer THan Expected
        [66]   // Sample Cone Dirty Alarm (Density is not 1)
        [14]   // Solution fill time exceeded Tank 1
        [33]   // XRF HW Watchdog Timeout
        [24]   // Hopper Levels Not OK at the Start Alarm
        [25]   // Check Tank diagnostics
        [42]   // Valve Module Comm Loss
        [43]   // DO_PH module Comm Loss
        [68]   // Water Supply Line Leak
        [27]   // Spare
        [28]   // Spare
        [13]   // Tank 10 Offline Alarm
        [2]   // No Available Tank Alarm
        [51]   // Tank 11 Offline Alarm
        [52]   // Tank 12 Offline Alarm
        [53]   // Tank 13 Offline Alarm
        [3]   // Purge Water Flow Low CNT reached
        [45]   // Spare
        [41]   // XRF Instrument Not fully in workstation
        [46]   // Spare
        [54]   // Tank 14 Offline Alarm
        [55]   // Tank 15 Offline Alarm
        [34]   // XRF Interlock Lid or E-stop
        [47]   // Spare
        [48]   // Spare
        [49]   // Spare
        [50]   // Spare
        [73]   // Spare
        [74]   // Spare
        [75]   // Spare
        [76]   // Spare
        [77]   // Spare
        [78]   // Spare
        [79]   // Spare
        [56]   // Tank 16 Offline Alarm
        [0]   // Low Air Pressure Alarm
        [10]   // Tank 7 Offline Alarm
        [38]   // XRF No Counts In Spectrum
        [63]   // Laser Compartment Dirty Alarm
        [11]   // Tank 8 Offline Alarm
        [12]   // Tank 9 Offline Alarm
        [30]   // XRF HW Error
        [15]   // Solution fill time exceeded Tank 2
        [16]   // Solution fill time exceeded Tank 3
        [17]   // Solution fill time exceeded Tank 4
        [18]   // Solution fill time exceeded Tank 5
        [19]   // Solution fill time exceeded Tank 6
        [20]   // Solution fill time exceeded Tank 7
        [21]   // Solution fill time exceeded Tank 8
        [22]   // Solution fill time exceeded Tank 9
        [23]   // Solution fill time exceeded Tank 10
        [58]   // Solution fill time exceeded Tank 12
        [59]   // Solution fill time exceeded Tank 13
        [60]   // Solution fill time exceeded Tank 14
        [61]   // Solution fill time exceeded Tank 15
        [4]   // Tank 1 Offline Alarm
        [5]   // Tank 2 Offline Alarm
        [6]   // Tank 3 Offline Alarm
        [31]   // XRF User Abort
        [7]   // Tank 4 Offline Alarm
        [62]   // Solution fill time exceeded Tank 16
        [1]   // Purge Water Flow Alarm
        [71]   // Line Leak
        [8]   // Tank 5 Offline Alarm
        [35]   // XRF Proximity Failure (Air Shoot)
        [44]   // XRF Window Dirity alarm
        [32]   // XRF Trigger Released
        [9]   // Tank 6 Offline Alarm
        [29]   // XRF heartbeat fault
        [40]   // XRF Proximity Abort
        [64]   // Sample Line Blocked
        [69]   // Pegged Screen Alarm
        [65]   // Sample Line Break
        [37]   // XRF No longer Needed
        [72]   // XRF door opened
        [67]   // Valve Maintenance Request Alarm
        [36]   // XRF External Interlock Abort
        [70]   // Laser High Fluctuation Alarm
        [57]   // Solution fill time exceeded Tank 11
        [26]   // Laser +-1% Error
   CS_CarbonSP : REAL := 100.0;
   CS_DINTParams : DINT[100] := ([0] := 12, [2] := 6, [4] := 40, [5] := 30, [6] := 30, [7] := 30, [8] := 30, [9] := 60, [10] := 10, [12] := 1, [13] := 5, [15] := 40, [16] := 5, [18] := 7, [19] := 10, [20] := 8, [21] := 10, [22] := 9, [23] := 10, [24] := 10, [25] := 10, [26] := 11, [27] := 10, [28] := 12, [29] := 10, [30] := 13, [31] := 10, [32] := 14, [33] := 10, [34] := 15, [35] := 10, [36] := 16, [37] := 10, [38] := 1, [40] := 60, [41] := 45, [42] := 45, [44] := 1, [48] := 1, [49] := 1, [50] := 1, [51] := 1, [52] := 1, [53] := 1, [54] := 1, [55] := 1, [56] := 1, [57] := 1, [58] := 1, [59] := 1, [66] := 492, [67] := 10, [75] := 5, [76] := 60, [77] := 1, [79] := 50, [80] := 10, [82] := 30, [84] := 1, [85] := 4,
        [86] := 5, [88] := 3, [92] := 33, [93] := 603992161, [97] := 1023, [98] := 1, [99] := -1205861878);
        [87]   // Auto start timer
        [92].6   // Auto Start Toggle 1= Enabled.
        [7]   // Activated Carbon Measurement Discharge Wash Time
        [93].15   // XRF bath wash sequence Xv15 open request
        [9]   // Activated Carbon Measurement Laser Stablise Time
        [6]   // Activated Carbon Measurement Screen (Measurement Cylnder) Wash Time Before Sample
        [93].0   // Flow switch or Floweter. Flow Switch = 1, Flowmeter = 0
        [82]   // Discharge Final Flushing Time (s) (Step 3)
        [67]   // Auto level calibration time remaining (s)
        [17]   // Last Tank Reached Delay Time (sec)
        [81]   // Discharge Valve Delay Time (sec) (Step 2)
        [93].24   // Water Supply 0 = MK5 no split, 1= MK6 Split
        [92].2   // XRF Power overide 1= POWER OFF
        [93].16   // Airshot positive pressure toggle Run at all times when enabled 1=enable
        [11]   // Activated Carbon Measurement Supply Tank Selection (0-10)
        [12]   // Activated Carbon Measurement Pulp Density Sample Tank
        [93].5   // Discharge Initial Flush Enable/Disabel
        [99].21   // 0 = Continuous Run After Schdule Sample, 1 = Idle After Schedule Sample
        [99].15   // XRF Measurement 1= Enable 0 = Disable
        [99].29   // 0 = Not All in Auto 1 = All in Auto
        [92].4   // HMI Stop has been requested. 1= true
        [93].1   // XRF Carbon Batch Test Sequence Start
        [80]   // Discharge Initial Flushing Time (s) (Step 1)
        [43].1   // Tank 2 Over filled
        [43].2   // Tank 3 Over filled
        [43].3   // Tank 4 Over filled
        [49]   // Transfer Pump 1 Run on Time
        [50]   // Transfer Pump 2 Run on Time
        [51]   // Transfer Pump 3 Run on Time
        [52]   // Transfer Pump 4 Run on Time
        [53]   // Transfer Pump 5 Run on Time
        [77]   // XRF Batch Water Test Cycles Requested
        [43].4   // Tank 5 Over filled
        [54]   // Transfer Pump 6 Run on Time
        [5]   // Activated Carbon Measurement Screen (Measuring Cylinder) Wash After Time
        [55]   // Transfer Pump 7 Run on Time
        [56]   // Transfer Pump 8 Run on Time
        [57]   // Transfer Pump 9 Run on Time
        [96].1   // Transfer Pump 1 Run Req
        [96].2   // Transfer Pump 2 Run Req
        [40]   // Manual Sample Purge Time
        [41]   // Manual Sample Drain Time
        [43].10   // Tank 11 Overfilled
        [43].11   // Tank 12 Overfilled
        [43].12   // Tank 13 Overfilled
        [43].13   // Tank 14 Overfilled
        [43].14   // Tank 15 Overfilled
        [43]   // Over Fill Cone Alarms
        [43].0   // Tank1 Over filled
        [96]   // Transfer Pump request
        [43].15   // Tank 16 Overfilled
        [92].1   // XRF reboot 1= reboot
        [42]   // Manual Sample Wash Time
        [96].3   // Transfer Pump 3 Run Req
        [97].10   // Schedule 1 Run Cmd
        [43].5   // Tank 6 Over filled
        [97].11   // Schedule 2 Run Cmd
        [97].12   // Schedule 3 Run Cmd
        [43].9   // Tank 10 Over filled
        [46]   // Step Time Remaining Min
        [97].0   // Schedule 1 Enable
        [97].13   // Schedule 4 Run Cmd
        [96].4   // Transfer Pump 4 Run Req
        [47]   // Step Time Remaining Sec
        [97].1   // Schedule 2 Enable
        [99].18   // 16 Tank enable disable 0 = 10, 1=16
        [19]   // Schdule 1 Min
        [97].14   // Schedule 5 Run Cmd
        [97].2   // Schedule 3 Enable
        [93].18   // XRF Batch Water Run Final Cycle
        [89]   // RunID
        [90]   // Spare
        [91]   // Spare
        [97].3   // Schedule 4 Enable
        [8]   // Activated Carbon Measurement Potable Water Rinse Time
        [43].6   // Tank 7 Over filled
        [21]   // Schdule 2 Min
        [23]   // Schdule 3 Min
        [96].5   // Transfer Pump 5 Run Req
        [43].7   // Tank 8 Over filled
        [92]   // CS BOOLS
        [25]   // Schdule 4 Min
        [18]   // Schdule 1 Hr
        [27]   // Schdule 5 Min
        [20]   // Schdule 2 Hr
        [22]   // Schdule 3 Hr
        [24]   // Schdule 4 Hr
        [29]   // Schdule 6 Min
        [1]   // Seq Timer in Sec
        [26]   // Schdule 5 Hr
        [93].10   // XRF Carbon Batch Test Sequence Running
        [43].8   // Tank 9 Over filled
        [97].15   // Schedule 6 Run Cmd
        [28]   // Schdule 6 Hr
        [30]   // Schdule 7 Hr
        [97].16   // Schedule 7 Run Cmd
        [93].25   // Tank Manual Changes
        [48]   // Transfer Feed Pump Run on Time
        [93].28   // CS Sample Seq Apply
        [93].8   // XRF Auto sequence batch water run completed
        [99].1   // 0 = Periodic Sample, 1 = Continuous Samlple
        [99].31   // Automatic Carbon Flow Enable/Dsiable
        [93].31   // CS Discharge Enable
        [99].8   // 1= Repeat Done 0 = Repeat Not Needed
        [93].7   // XRF auto test started
        [97].4   // Schedule 5 Enable
        [96].11   // Transfer Pump Discharge Run Req
        [99].6   // Dilution Enable 0 = Disable, 1= Enable
        [37]   // Schdule 10 Min
        [70]   // XRF Beam 1 Min
        [71]   // XRF Beam 1 Max
        [99].28   // Initial Purge Enable 0 = disable 1=enable
        [13]   // Activated Carbon Measurement Pulp Density Sample Time (sec)
        [96].6   // Transfer Pump 6 Run Req
        [93].12   // XRF Button Visability. Stop. 1=visable
        [93].11   // XRF Button Visability. Start. 1=visable
        [93].13   // XRF Button Visability. Power 1=visable
        [93].20   // XRF Carbon Batch Test Sequence Running
        [45]   // Step Time Remaining Hr
        [97].5   // Schedule 6 Enable
        [93].2   // XRF Carbon Batch Test Sequence Latch
        [97]   // Schedules
        [32]   // Schdule 8 Hr
        [93].27   // Sample Isolation valve 1= enable 0= disable
        [79]   // XRF Cooling Temp limit
        [10]   // Activated Carbon Measurement Drain Time
        [99].13   // Density 1= Enabled 0 = Disabled
        [15]   // Activated Carbon Measurment DO and pH stablising time (sec)
        [93].9   // XRF Auto sequence batch water run skip required
        [99].16   // Cyanide Measurement 1= Enabled 0 = Disabled
        [39]   // Manual Sample Tank 0 - 9 0 = Tank1, 15 = Tank 16
        [3]   // Activated Carbon Measurement Cycle Time Period Setpoint (Min)
        [99].25   // Program Pause Request 0 = resume, 1 = Pause
        [31]   // Schdule 7 Min
        [92].3   // PC Power overide 1= POWER OFF
        [99]   // CS BOOLS
        [99].2   // Step 1 Permisssive 0 = not OK to Proceed 1= OK to proceed
        [97].17   // Schedule 8 Run Cmd
        [34]   // Schdule 9 Hr
        [99].3   // DO and pH Enable 0 = Disable, 1 = Enable Always enabled
        [98].14   // Wash
        [96].7   // Transfer Pump 7 Run Req
        [84]   // Second Result view 0 - g/L 1 - Slurry VOL (L) 2 - Carbon Mass (g) 3 - Carbon Volume (mL) 4 - DO (ppm) 5 - pH 6 - CN (ppm) 7 - ml/L 8 - Slurry weight (kg) 9 - ORP (mv) 10 - Temperature pH ('C) 11 - Temperature DO ('C) 12 - Carbon Height (mm) 13 - Flow rate (L/s) 14 - Fill time (s) 15 - Purge water used (L) 16 - Sample duration (s) 17-Density 18-Au
        [95]   // Transfer pump running Feedback
        [97].9   // Schedule 10 Enable
        [93].23   // Water selection 1 = Process 0 = Potable
        [96].8   // Transfer Pump 8 Run Req
        [96].9   // Transfer Pump 9 Run Req
        [93].30   // CS Booster Enable
        [99].24   // Tank Select Apply Bit
        [97].6   // Schedule 7 Enable
        [99].14   // Airshot 1= Enabled 0 = Disabled
        [93].17   // Solution fill time out skip
        [97].19   // Schedule 10 Run Cmd
        [99].9   // Low Air Pressure Enable
        [97].7   // Schedule 8 Enable
        [97].8   // Schedule 9 Enable
        [72]   // XRF Beam 2 Min
        [74]   // Zero XRF readings
        [99].19   // XRF Power Button
        [73]   // XRF Beam 2 Max
        [98].11   // Bucket In place
        [93]   // CS BOOLS Additional
        [99].20   // Reset Records
        [99].23   // OnceBatch Bit
        [93].22   // Pruge Required
        [99].7   // Sample Error Flag
        [93].6   // XRF booting flag
        [98]   // Manual Sample Tank Selections
        [94]   // Transfer Pump Path
        [97].18   // Schedule 9 Run Cmd
        [99].30   // All to Auto
        [98].12   // Manual Sample Purge
        [33]   // Schdule 8 Min
        [99].26   // Add Water 5L
        [35]   // Schdule 9 Min
        [0]   // Step_intlk OR Permissive Indicator
        [66]   // Sample Duration in Seccccc
        [36]   // Schdule 10 Hr
        [99].0   // Time Change Apply BTN
        [38]   // Tank Choose
        [14]   // CS Last Sampling Tank Indicator
        [96].0   // Transfer Feed Pump Run Req
        [93].3   // XRF Power button push delay
        [96].10   // Transfer Pump 10 Run Req
        [58]   // Transfer Pump 10 Run on Time
        [60]   // Transfer Pump 11 Run On Time
        [99].22   // Only One Tank Available
        [99].5   // Bottom Wash Trigger XV 15
        [93].19   // XRF Batch Water Run Cycling
        [98].0   // Manual sample Tank 1
        [98].1   // Manual sample Tank 2
        [93].26   // 1= FTP 0 = Email data files
        [98].2   // Manual sample Tank 3
        [98].3   // Manual sample Tank 4
        [98].4   // Manual sample Tank 5
        [98].5   // Manual sample Tank 6
        [98].6   // Manual sample Tank 7
        [98].7   // Manual sample Tank 8
        [98].8   // Manual sample Tank 9
        [98].13   // Manual sample Drain
        [99].4   // Purge Trigger XV 11
        [98].16   // Manual Result Sync override
        [98].9   // Manual sample Tank 10
        [61]   // Transfer Pump 12 Run On Time
        [62]   // Transfer Pump 13 Run On Time
        [63]   // Transfer Pump 14 Run On Time
        [64]   // Transfer Pump 15 Run On Time
        [65]   // Transfer Pump 16 Run On Time
        [93].14   // XRF results moved flag
        [93].29   // CS Sample Seq Cal Done
        [98].15   // Manual Sample Override
        [99].27   // Radar Calibration Done
        [4]   // Activated Carbon Measurement Sample Cone Wash Time
        [2]   // CS Current Sampling Tank Indicator
        [92].0   // XRF power enable 1=power on
        [59]   // Transfer Pump Discharge Run On Time
        [75]   // XRF Batch Water Test Spray Time (s)
        [76]   // XRF Batch Water Test Delay Time (s)
        [78]   // XRF Batch Water Test Cycles Current
        [93].21   // Use Purge Water for cone fill
        [93].4   // FLow switch Input status 1=Flow
        [16]   // Sample Error Cnt
        [44]   // Email Num
        [98].10   // Manual Sample Run
        [99].11   // Schedule Run Enable 0 = Disable 1 = Enable
        [99].12   // Manual Sample Enable 0 = Disable 1= Enable
        [99].17   // Apply Liquid and solid density to all tank
        [99].10   // Last Tank Reached
        [68]   // XRF Dirty Window Setpoint (ppm Ca Raw)
        [69]   // XRF Dirty Window Number of delay cycles
        [92].8   // Debounce Timer Running Hold Valve Open
        [88]   // Sample DB timer Sec
        [83]   // First Result view 0 - g/L 1 - Slurry VOL (L) 2 - Carbon Mass (g) 3 - Carbon Volume (mL) 4 - DO (ppm) 5 - pH 6 - CN (ppm) 7 - ml/L 8 - Slurry weight (kg) 9 - ORP (mv) 10 - Temperature pH ('C) 11 - Temperature DO ('C) 12 - Carbon Height (mm) 13 - Flow rate (L/s) 14 - Fill time (s) 15 - Purge water used (L) 16 - Sample duration (s) 17-Density 18-Au
        [85]   // Third Result view 0 - g/L 1 - Slurry VOL (L) 2 - Carbon Mass (g) 3 - Carbon Volume (mL) 4 - DO (ppm) 5 - pH 6 - CN (ppm) 7 - ml/L 8 - Slurry weight (kg) 9 - ORP (mv) 10 - Temperature pH ('C) 11 - Temperature DO ('C) 12 - Carbon Height (mm) 13 - Flow rate (L/s) 14 - Fill time (s) 15 - Purge water used (L) 16 - Sample duration (s) 17-Density 18-Au
        [86]   // Forth Result view 0 - g/L 1 - Slurry VOL (L) 2 - Carbon Mass (g) 3 - Carbon Volume (mL) 4 - DO (ppm) 5 - pH 6 - CN (ppm) 7 - ml/L 8 - Slurry weight (kg) 9 - ORP (mv) 10 - Temperature pH ('C) 11 - Temperature DO ('C) 12 - Carbon Height (mm) 13 - Flow rate (L/s) 14 - Fill time (s) 15 - Purge water used (L) 16 - Sample duration (s) 17-Density 18-Au
        [92].5   // XRF software WatchDog 10 minuts then move on and triger reboot
   CS_EventNum : DINT := 1;
   CS_REALParams : REAL[80] := ([0] := 1410.0, [1] := 1447.2368, [4] := 16.0, [5] := 58.0, [6] := 0.5, [9] := 1.0, [10] := 35.0, [11] := 17.945206, [12] := 600.0, [13] := 1218.0, [14] := 814.0, [15] := -35.206055, [16] := 212.71796, [17] := 1306342.6, [18] := 293.39545, [19] := 272.0, [20] := 1023.1226, [21] := 3.4871795, [22] := 50.0, [23] := 10.0, [24] := 3786.0, [25] := 13615.0, [26] := 16000.0, [27] := 17086.0, [28] := 17670.0, [29] := 6.017242, [30] := 9.085448, [31] := 1410.0, [32] := 3789.0, [33] := 20.0, [46] := -10.52187, [47] := 418.39386, [48] := inf, [49] := 1.0, [50] := 2.83, [52] := 60.0, [53] := 1350.0, [56] := 1.15, [58] := 5.0, [59] := 10.0, [60] := 15.0, [61] := 20.0, [62] := 2791.0, [63] := 1482.59, [64] := 5.0);   // CS REAL Parameters
        [16]   // Activated Carbon Measurement Virtual Small Cone Height (mm)
        [52]   // XRF - Bottom of strainer to top of window distance. (mm)
        [11]   // Activated Carbon Measurement Sample Cone Volume Actual (Litres)
        [17]   // Activated Carbon Measurement Cyclinder Volume
        [20]   // Activated Carbon Measurement Measured Height After Cylinder (mm)
        [0]   // Activated Carbon Measurement Empty Distance
        [6]   // Activated Carbon Measurement Sample Carbon Specific Gravity
        [9]   // Activated Carbon Measurement Minimum Acceptable Result Value
        [10]   // Activated Carbon Measurement Maximum Acceptable Result Value
        [5]   // Activated Carbon Measurement Cylinder Cross Sectional Diameter (mm)
        [12]   // Activated Carbon Measurement Strainer Cone Diameter (mm)
        [15]   // Activated Carbon Measurement Measured Height (mm)
        [1]   // Activated Carbon Measurement Full Distance
        [23]   // Potable Water Fill SP at the end of Step
        [14]   // Activated Carbon Measurement Strainer Cylinder Height (mm)
        [18]   // Activated Carbon Measurement Diameter After Cylinder (mm)
        [4]   // Activated Carbon Measurement Sample Cone Setpoint (Litres)
        [26]   // Cone Level Raw at 10 L
        [27]   // Cone Level Raw at 15 L
        [2]   // Activated Carbon Measurement Empty Distance (Redundant)
        [28]   // Cone Level Raw at 20 L
        [32]   // Cone Level Raw Reading
        [42]   // DO Partial Pressure Pa
        [45]   // Density - Empty Weight
        [54]   // Purge Volume in L Live
        [3]   // Activated Carbon Measurement Sample Cone Volume (Litres)
        [40]   // pH Reference Impedance ohms
        [55]   // Last Measured Water Density
        [39]   // pH Glass Impedance Mohms
        [36]   // pH rH
        [21]   // Activated Carbon Measurement Gradient = Height/Base
        [47]   // Density - Slurry Density
        [65]   // Spare
        [66]   // Spare
        [67]   // Spare
        [68]   // Spare
        [69]   // Spare
        [70]   // Spare
        [71]   // Spare
        [72]   // Spare
        [58]   // Cone Level First Point L
        [60]   // Cone Level Third Point L
        [61]   // Cone Level Forth Point L
        [35]   // pH probe Temp Degrees C
        [24]   // Cone Level Raw at 0 L
        [73]   // Spare
        [25]   // Cone Level Raw at 5 L
        [74]   // Spare
        [75]   // Spare
        [41]   // DO probe temp Degrees C
        [46]   // Density - Slurry Weight
        [76]   // Spare
        [77]   // Spare
        [78]   // Spare
        [79]   // Spare
        [31]   // Laser Level Maximum Scale
        [37]   // pH ORP %
        [48]   // Temp Sample filling rate L/sec
        [34]   // ORP mV
        [62]   // Spare
        [59]   // Cone Level Second Point L
        [19]   // Activated Carbon Measurement Cone Height (mm)
        [22]   // Activated Carbon Measurement % Allowable results
        [57]   // Laser Empty with Flap open
        [33]   // Max Solution Level
        [29]   // DO Live Reading
        [50]   // Density - Solid SG
        [7]   // Activated Carbon Measurement pH
        [49]   // Density - Liquid SG
        [38]   // pH Raw mV
        [13]   // Activated Carbon Measurement Strainer Full Height (mm)
        [44]   // DO raw value μs
        [30]   // pH Live Reading
        [43]   // DO saturation %
        [56]   // Last Water Density Compare
        [51]   // Result mL/L
        [53]   // XRF - Laser min distance calc. (mm)
        [8]   // Activated Carbon Measurement DO (ppm)
        [63]   // XRF Auto sequence carbon level store
   CS_Result : CS_Results := (Run_ID := 2791, Min := 3, Day := 22, Month := 11, Year := 2021, Sample_DO := 5.1741395, Sample_pH := 9.07387, Sample_VOL := 17.945206, Au := -93.0, Density := 418.39386, EmptyDist := 1410.0, FullDist := 1444.842, Slurry_Weight := -10.52187, Sample_Tank := 6, Carbon_Height := -35.206055, Sample_FlowRate := 1.812647, Sample_FillTime := 9.900001, SampleDuration := 707);   // Sample Result Live Async
   CS_Results : CS_Results[20] := ([1].Run_ID := 2783, [1].Hour := 22, [1].Min := 25, [1].Day := 21, [1].Month := 11, [1].Year := 2021, [1].Sample_DO := 5.78888, [1].Sample_pH := 9.147207, [1].Sample_VOL := 16.763699, [1].Density := 401.0287, [1].EmptyDist := 1410.0, [1].FullDist := 1447.1833, [1].ErrorFlag := 1, [1].Slurry_Weight := -10.52187, [1].Sample_Tank := 1, [1].Carbon_Height := -37.18335, [1].Sample_FlowRate := 0.23682894, [1].Sample_FillTime := 70.784, [1].SampleDuration := 1055, [2].Run_ID := 2761, [2].Carbon_VOL_ml := 175.5638, [2].Carbon_MASS := 87.7819, [2].Carbon_DIST := 5.193985, [2].Hour := 16, [2].Min := 28, [2].Day := 21, [2].Month := 11, [2].Year := 2021, [2].Sample_DO := 6.1882257, [2].Sample_pH := 9.219038, [2].Sample_VOL := 16.900684, [2].Density := 403.04202, [2].EmptyDist := 1410.0, [2].FullDist := 1343.5509, [2].Carbon_mLperL := 10.38797, [2].Slurry_Weight := -10.52187, [2].Sample_Tank := 2, [2].Carbon_Height := 66.4491, [2].Sample_FlowRate := 1.8778536, [2].Sample_FillTime := 9.000001, [2].DisplacedCarbonVol := 1560.5671, [2].DisplacedCarbonMass := 780.28357, [2].SampleDuration := 934, [3].Run_ID := 2785, [3].Hour := 22, [3].Min := 56, [3].Day := 21, [3].Month := 11, [3].Year := 2021, [3].Sample_DO := 5.975054, [3].Sample_pH := 9.085041, [3].Sample_VOL := 17.71404, [3].Density := 414.99634, [3].EmptyDist := 1410.0, [3].FullDist := 1441.737, [3].ErrorFlag := 1, [3].Slurry_Weight := -10.52187, [3].Sample_Tank := 3, [3].Carbon_Height := -31.73706, [3].Sample_FlowRate := 1.3902087,
        [3].Sample_FillTime := 12.742001, [3].SampleDuration := 926, [4].Run_ID := 2787, [4].Hour := 23, [4].Min := 27, [4].Day := 21, [4].Month := 11, [4].Year := 2021, [4].Sample_DO := 5.6127687, [4].Sample_pH := 9.112585, [4].Sample_VOL := 17.34589, [4].Density := 409.58542, [4].EmptyDist := 1410.0, [4].FullDist := 1447.225, [4].ErrorFlag := 1, [4].Slurry_Weight := -10.52187, [4].Sample_Tank := 4, [4].Carbon_Height := -37.224976, [4].Sample_FlowRate := 1.464777, [4].Sample_FillTime := 11.842001, [4].SampleDuration := 926, [5].Run_ID := 2789, [5].Carbon_VOL_ml := 64.33941, [5].Carbon_MASS := 32.169704, [5].Carbon_DIST := 1.8038509, [5].Hour := 23, [5].Min := 51, [5].Day := 21, [5].Month := 11, [5].Year := 2021, [5].Sample_DO := 5.7689, [5].Sample_pH := 9.094793, [5].Sample_VOL := 17.833904, [5].Density := 416.75797, [5].EmptyDist := 1410.0, [5].FullDist := 1385.6482, [5].ErrorFlag := 1, [5].Carbon_mLperL := 3.6077018, [5].Slurry_Weight := -10.52187, [5].Sample_Tank := 5, [5].Carbon_Height := 24.351807, [5].Sample_FlowRate := 1.3210299, [5].Sample_FillTime := 13.500001, [5].DisplacedCarbonVol := 476.58823, [5].DisplacedCarbonMass := 238.29411, [5].SampleDuration := 736, [6].Run_ID := 2790, [6].Min := 3, [6].Day := 22, [6].Month := 11, [6].Year := 2021, [6].Sample_DO := 5.1891594, [6].Sample_pH := 9.087861, [6].Sample_VOL := 17.893835, [6].Density := 417.63882, [6].EmptyDist := 1410.0, [6].FullDist := 1445.206, [6].Slurry_Weight := -10.52187, [6].Sample_Tank := 6, [6].Carbon_Height := -35.206055,
        [6].Sample_FlowRate := 1.8639408, [6].Sample_FillTime := 9.600001, [6].SampleDuration := 716, [7].Run_ID := 2779, [7].Hour := 21, [7].Min := 19, [7].Day := 21, [7].Month := 11, [7].Year := 2021, [7].Sample_DO := 5.578247, [7].Sample_pH := 9.083747, [7].Sample_VOL := 17.388699, [7].Density := 410.2146, [7].EmptyDist := 1410.0, [7].FullDist := 1445.2788, [7].ErrorFlag := 1, [7].Slurry_Weight := -10.52187, [7].Sample_Tank := 7, [7].Carbon_Height := -35.27881, [7].Sample_FlowRate := 1.7047743, [7].Sample_FillTime := 10.200001, [7].SampleDuration := 1025, [8].Run_ID := 2781, [8].Hour := 21, [8].Min := 52, [8].Day := 21, [8].Month := 11, [8].Year := 2021, [8].Sample_DO := 5.314984, [8].Sample_pH := 9.142456, [8].Sample_VOL := 17.465754, [8].Density := 411.34714, [8].EmptyDist := 1410.0, [8].FullDist := 1447.225, [8].ErrorFlag := 1, [8].Slurry_Weight := -10.52187, [8].Sample_Tank := 8, [8].Carbon_Height := -37.224976, [8].Sample_FlowRate := 2.0792563, [8].Sample_FillTime := 8.400001, [8].SampleDuration := 974);   // Results Just for DataStore
        [0]   // Zero
   CS_ResultsSync : CS_Results := (Run_ID := 2791, Min := 3, Day := 22, Month := 11, Year := 2021, Sample_DO := 5.1891594, Sample_pH := 9.087861, Sample_VOL := 17.893835, Density := 417.63882, EmptyDist := 1410.0, FullDist := 1445.206, ErrorFlag := 1, Slurry_Weight := -10.52187, Sample_Tank := 6, Carbon_Height := -35.206055, Sample_FlowRate := 1.8639408, Sample_FillTime := 9.600001, SampleDuration := 707);
   CS_ResultStore : CS_Results[20,20] := ([0,0].Carbon_MASS := 243.40945, [0,0].Carbon_DIST := 121.70473, [0,0].Hour := 1091385754, [0,0].Min := 10, [0,0].Day := 6, [0,0].Month := 28, [0,0].Year := 10, [0,0].Sample_DO := 2.83e-42, [0,0].Sample_pH := 0.009032038, [0,0].Sample_VOL := 9.623773, [0,0].Au := 13.788462, [0,0].FullDist := 816.0, [0,0].ErrorFlag := 1143800342, [0,1].Carbon_MASS := 271.58386, [0,1].Carbon_DIST := 135.79193, [0,1].Hour := 1092380803, [0,1].Min := 9, [0,1].Day := 27, [0,1].Month := 28, [0,1].Year := 10, [0,1].Sample_DO := 2.83e-42, [0,1].Sample_pH := 0.009110672, [0,1].Sample_VOL := 9.632538, [0,1].Au := 13.891025, [0,1].FullDist := 816.0, [0,1].ErrorFlag := 1143565246, [0,2].Carbon_MASS := 353.7815, [0,2].Carbon_DIST := 176.89075, [0,2].Hour := 1095397470, [0,2].Min := 8, [0,2].Day := 47, [0,2].Month := 28, [0,2].Year := 10, [0,2].Sample_DO := 2.83e-42, [0,2].Sample_pH := 0.009201728, [0,2].Sample_VOL := 9.640686, [0,2].Au := 13.980769, [0,2].FullDist := 816.0, [0,2].ErrorFlag := 1142879364, [0,3].Carbon_MASS := 374.80103, [0,3].Carbon_DIST := 187.40051, [0,3].Hour := 1095772877, [0,3].Min := 8, [0,3].Day := 8, [0,3].Month := 28, [0,3].Year := 10, [0,3].Sample_DO := 2.83e-42, [0,3].Sample_pH := 0.009260239, [0,3].Sample_VOL := 9.647568, [0,3].Au := 14.403847, [0,3].FullDist := 816.0, [0,3].ErrorFlag := 1142703971, [0,4].Carbon_MASS := 382.55075, [0,4].Carbon_DIST := 191.27538, [0,4].Hour := 1096443523, [0,4].Min := 7, [0,4].Day := 29, [0,4].Month := 28, [0,4].Year := 10, [0,4].Sample_DO := 2.83e-42,
        [0,4].Sample_pH := 0.00928737, [0,4].Sample_VOL := 9.646709, [0,4].Au := 14.01282, [0,4].FullDist := 816.0, [0,4].ErrorFlag := 1142639305, [0,5].Carbon_MASS := 478.19553, [0,5].Carbon_DIST := 239.09776, [0,5].Hour := 1099387770, [0,5].Min := 6, [0,5].Day := 50, [0,5].Month := 28, [0,5].Year := 10, [0,5].Sample_DO := 2.83e-42, [0,5].Sample_pH := 0.009283138, [0,5].Sample_VOL := 9.650078, [0,5].Au := 14.134615, [0,5].FullDist := 816.0, [0,5].ErrorFlag := 1141841216, [0,6].Carbon_MASS := 449.23972, [0,6].Carbon_DIST := 224.61986, [0,6].Hour := 1098726111, [0,6].Min := 6, [0,6].Day := 7, [0,6].Month := 28, [0,6].Year := 10, [0,6].Sample_DO := 2.83e-42, [0,6].Sample_pH := 0.009290737, [0,6].Sample_VOL := 9.636368, [0,6].Au := 14.192308, [0,6].FullDist := 816.0, [0,6].ErrorFlag := 1142082832, [0,7].Carbon_MASS := 463.65625, [0,7].Carbon_DIST := 231.82812, [0,7].Hour := 1099196831, [0,7].Min := 5, [0,7].Day := 27, [0,7].Month := 28, [0,7].Year := 10, [0,7].Sample_DO := 2.83e-42, [0,7].Sample_pH := 0.009273029, [0,7].Sample_VOL := 9.623397, [0,7].Au := 14.006411, [0,7].FullDist := 816.0, [0,7].ErrorFlag := 1141962536, [0,8].Carbon_MASS := 465.50067, [0,8].Carbon_DIST := 232.75034, [0,8].Hour := 1099179823, [0,8].Min := 4, [0,8].Day := 48, [0,8].Month := 28, [0,8].Year := 10, [0,8].Sample_DO := 2.83e-42, [0,8].Sample_pH := 0.009282848, [0,8].Sample_VOL := 9.619032, [0,8].Au := 14.089743, [0,8].FullDist := 816.0, [0,8].ErrorFlag := 1141947146, [0,9].Carbon_MASS := 465.315, [0,9].Carbon_DIST := 232.6575, [0,9].Hour := 1099215936,
        [0,9].Min := 4, [0,9].Day := 9, [0,9].Month := 28, [0,9].Year := 10, [0,9].Sample_DO := 2.83e-42, [0,9].Sample_pH := 0.009250989, [0,9].Sample_VOL := 9.6214, [0,9].Au := 14.0256405, [0,9].FullDist := 816.0, [0,9].ErrorFlag := 1141948695, [0,10].Carbon_MASS := 445.2612, [0,10].Carbon_DIST := 222.6306, [0,10].Hour := 1098917895, [0,10].Min := 3, [0,10].Day := 30, [0,10].Month := 28, [0,10].Year := 10, [0,10].Sample_DO := 2.83e-42, [0,10].Sample_pH := 0.009255391, [0,10].Sample_VOL := 9.620493, [0,10].Au := 13.897436, [0,10].FullDist := 816.0, [0,10].ErrorFlag := 1142116030, [0,11].Carbon_MASS := 418.47186, [0,11].Carbon_DIST := 209.23593, [0,11].Hour := 1097917500, [0,11].Min := 2, [0,11].Day := 50, [0,11].Month := 28, [0,11].Year := 10, [0,11].Sample_DO := 2.83e-42, [0,11].Sample_pH := 0.009251575, [0,11].Sample_VOL := 9.629539, [0,11].Au := 13.897436, [0,11].FullDist := 816.0, [0,11].ErrorFlag := 1142339568, [0,12].Carbon_MASS := 397.9465, [0,12].Carbon_DIST := 198.97325, [0,12].Hour := 1096972028, [0,12].Min := 2, [0,12].Day := 11, [0,12].Month := 28, [0,12].Year := 10, [0,12].Sample_DO := 2.83e-42, [0,12].Sample_pH := 0.009289178, [0,12].Sample_VOL := 9.620131, [0,12].Au := 14.057692, [0,12].FullDist := 816.0, [0,12].ErrorFlag := 1142510838, [0,13].Carbon_MASS := 439.47293, [0,13].Carbon_DIST := 219.73647, [0,13].Hour := 1098725086, [0,13].Min := 1, [0,13].Day := 32, [0,13].Month := 28, [0,13].Year := 10, [0,13].Sample_DO := 2.83e-42, [0,13].Sample_pH := 0.009294648, [0,13].Sample_VOL := 9.625267, [0,13].Au := 13.884615,
        [0,13].FullDist := 816.0, [0,13].ErrorFlag := 1142164329, [0,14].Carbon_MASS := 465.3229, [0,14].Carbon_DIST := 232.66145, [0,14].Hour := 1099200213, [0,14].Day := 53, [0,14].Month := 28, [0,14].Year := 10, [0,14].Sample_DO := 2.83e-42, [0,14].Sample_pH := 0.0092815, [0,14].Sample_VOL := 9.624359, [0,14].Au := 14.051282, [0,14].FullDist := 816.0, [0,14].ErrorFlag := 1141948629, [0,15].Carbon_MASS := 367.86093, [0,15].Carbon_DIST := 183.93047, [0,15].Hour := 1095800104, [0,15].Day := 13, [0,15].Month := 28, [0,15].Year := 10, [0,15].Sample_DO := 2.83e-42, [0,15].Sample_pH := 0.009287097, [0,15].Sample_VOL := 9.626813, [0,15].Au := 14.108975, [0,15].FullDist := 816.0, [0,15].ErrorFlag := 1142761881, [0,16].Carbon_MASS := 401.65323, [0,16].Carbon_DIST := 200.82661, [0,16].Hour := 1097049045, [0,16].Min := 23, [0,16].Day := 34, [0,16].Month := 27, [0,16].Year := 10, [0,16].Sample_DO := 2.83e-42, [0,16].Sample_pH := 0.009269633, [0,16].Sample_VOL := 9.617054, [0,16].Au := 14.115385, [0,16].FullDist := 816.0, [0,16].ErrorFlag := 1142479908, [0,17].Carbon_MASS := 457.60718, [0,17].Carbon_DIST := 228.80359, [0,17].Hour := 1099138846, [0,17].Min := 22, [0,17].Day := 55, [0,17].Month := 27, [0,17].Year := 10, [0,17].Sample_DO := 2.83e-42, [0,17].Sample_pH := 0.009253993, [0,17].Sample_VOL := 9.615788, [0,17].Au := 13.916667, [0,17].FullDist := 816.0, [0,17].ErrorFlag := 1142013011, [0,18].Carbon_MASS := 404.1081, [0,18].Carbon_DIST := 202.05405, [0,18].Hour := 1097539088, [0,18].Min := 22, [0,18].Day := 15, [0,18].Month := 27, [0,18].Year := 10, [0,18].Sample_DO := 2.83e-42,
        [0,18].Sample_pH := 0.009211945, [0,18].Sample_VOL := 9.60799, [0,18].Au := 13.75, [0,18].FullDist := 816.0, [0,18].ErrorFlag := 1142459424, [0,19].Carbon_MASS := 406.75348, [0,19].Carbon_DIST := 203.37674, [0,19].Hour := 1097582328, [0,19].Min := 21, [0,19].Day := 36, [0,19].Month := 27, [0,19].Year := 10, [0,19].Sample_DO := 2.83e-42, [0,19].Sample_pH := 0.009202228, [0,19].Sample_VOL := 9.608318, [0,19].Au := 13.801282, [0,19].FullDist := 816.0, [0,19].ErrorFlag := 1142437350, [1,0].Run_ID := 2783, [1,0].Hour := 22, [1,0].Min := 25, [1,0].Day := 21, [1,0].Month := 11, [1,0].Year := 2021, [1,0].Sample_DO := 5.78888, [1,0].Sample_pH := 9.147207, [1,0].Sample_VOL := 16.763699, [1,0].Density := 401.0287, [1,0].EmptyDist := 1410.0, [1,0].FullDist := 1447.1833, [1,0].ErrorFlag := 1, [1,0].Slurry_Weight := -10.52187, [1,0].Sample_Tank := 1, [1,0].Carbon_Height := -37.18335, [1,0].Sample_FlowRate := 0.23682894, [1,0].Sample_FillTime := 70.784, [1,0].SampleDuration := 1055, [1,1].Run_ID := 2782, [1,1].Hour := 22, [1,1].Min := 9, [1,1].Day := 21, [1,1].Month := 11, [1,1].Year := 2021, [1,1].Sample_DO := 5.3873496, [1,1].Sample_pH := 9.17127, [1,1].Sample_VOL := 16.215754, [1,1].Density := 392.9753, [1,1].EmptyDist := 1410.0, [1,1].FullDist := 1438.2352, [1,1].Slurry_Weight := -10.52187, [1,1].Sample_Tank := 1, [1,1].Carbon_Height := -28.23523, [1,1].Sample_FlowRate := 0.08818469, [1,1].Sample_FillTime := 183.884, [1,1].SampleDuration := 975, [1,2].Run_ID := 2769, [1,2].Hour := 18, [1,2].Min := 56, [1,2].Day := 21, [1,2].Month := 11,
        [1,2].Year := 2021, [1,2].Sample_DO := 5.83768, [1,2].Sample_pH := 9.173825, [1,2].Sample_VOL := 16.686644, [1,2].Density := 399.89615, [1,2].EmptyDist := 1410.0, [1,2].FullDist := 1440.8074, [1,2].ErrorFlag := 1, [1,2].Slurry_Weight := -10.52187, [1,2].Sample_Tank := 1, [1,2].Carbon_Height := -30.807373, [1,2].Sample_FlowRate := 0.13854505, [1,2].Sample_FillTime := 120.442, [1,2].SampleDuration := 1015, [1,3].Run_ID := 2768, [1,3].Hour := 18, [1,3].Min := 40, [1,3].Day := 21, [1,3].Month := 11, [1,3].Year := 2021, [1,3].Sample_DO := 5.7754235, [1,3].Sample_pH := 9.192625, [1,3].Sample_VOL := 16.061644, [1,3].Density := 390.71027, [1,3].EmptyDist := 1410.0, [1,3].FullDist := 1437.6216, [1,3].Slurry_Weight := -10.52187, [1,3].Sample_Tank := 1, [1,3].Carbon_Height := -27.621582, [1,3].Sample_FlowRate := 0.10948633, [1,3].Sample_FillTime := 146.7, [1,3].SampleDuration := 973, [1,4].Run_ID := 2763, [1,4].Hour := 17, [1,4].Min := 11, [1,4].Day := 21, [1,4].Month := 11, [1,4].Year := 2021, [1,4].Sample_DO := 5.7825546, [1,4].Sample_pH := 9.13574, [1,4].Sample_VOL := 16.344177, [1,4].Density := 394.8628, [1,4].EmptyDist := 1410.0, [1,4].FullDist := 1447.0728, [1,4].ErrorFlag := 1, [1,4].Slurry_Weight := -10.52187, [1,4].Sample_Tank := 1, [1,4].Carbon_Height := -37.072754, [1,4].Sample_FlowRate := 0.24763905, [1,4].Sample_FillTime := 66.0, [1,4].SampleDuration := 1602, [1,5].Run_ID := 2762, [1,5].Hour := 16, [1,5].Min := 58, [1,5].Day := 21, [1,5].Month := 11, [1,5].Year := 2021, [1,5].Sample_DO := 6.393456, [1,5].Sample_pH := 9.164372, [1,5].Sample_VOL := 10.418968,
        [1,5].Density := 307.77722, [1,5].EmptyDist := 1410.0, [1,5].FullDist := 1447.0728, [1,5].Slurry_Weight := -10.52187, [1,5].Sample_Tank := 1, [1,5].Carbon_Height := -37.072754, [1,5].Sample_FlowRate := 0.052068803, [1,5].Sample_FillTime := 200.1, [1,5].SampleDuration := 872, [1,6].Run_ID := 2760, [1,6].Hour := 16, [1,6].Min := 13, [1,6].Day := 21, [1,6].Month := 11, [1,6].Year := 2021, [1,6].Sample_DO := 5.364569, [1,6].Sample_pH := 9.1462965, [1,6].Sample_VOL := 16.275684, [1,6].Density := 393.8561, [1,6].EmptyDist := 1410.0, [1,6].FullDist := 1427.1587, [1,6].ErrorFlag := 1, [1,6].Slurry_Weight := -10.52187, [1,6].Sample_Tank := 1, [1,6].Carbon_Height := -17.158691, [1,6].Sample_FlowRate := 0.24112125, [1,6].Sample_FillTime := 67.5, [1,6].SampleDuration := 974, [1,7].Run_ID := 2759, [1,7].Carbon_VOL_ml := 3.8225007, [1,7].Carbon_MASS := 1.9112504, [1,7].Carbon_DIST := 0.11602601, [1,7].Hour := 15, [1,7].Min := 58, [1,7].Day := 21, [1,7].Month := 11, [1,7].Year := 2021, [1,7].Sample_DO := 5.32723, [1,7].Sample_pH := 9.180892, [1,7].Sample_VOL := 16.472603, [1,7].Density := 396.7503, [1,7].EmptyDist := 1410.0, [1,7].FullDist := 1408.5532, [1,7].Carbon_mLperL := 0.23205201, [1,7].Slurry_Weight := -10.52187, [1,7].Sample_Tank := 1, [1,7].Carbon_Height := 1.4467773, [1,7].Sample_FlowRate := 0.1562243, [1,7].Sample_FillTime := 105.442, [1,7].DisplacedCarbonVol := 2.900173, [1,7].DisplacedCarbonMass := 1.4500865, [1,7].SampleDuration := 974, [1,8].Run_ID := 2744, [1,8].Carbon_VOL_ml := 36.00317, [1,8].Carbon_MASS := 18.001585, [1,8].Carbon_DIST := 1.1072065, [1,8].Hour := 12, [1,8].Min := 16, [1,8].Day := 21, [1,8].Month := 11,
        [1,8].Year := 2021, [1,8].Sample_DO := 5.4306774, [1,8].Sample_pH := 9.17495, [1,8].Sample_VOL := 16.258562, [1,8].Density := 393.60446, [1,8].EmptyDist := 1410.0, [1,8].FullDist := 1396.3732, [1,8].ErrorFlag := 1, [1,8].Carbon_mLperL := 2.214413, [1,8].Slurry_Weight := -10.52187, [1,8].Sample_Tank := 1, [1,8].Carbon_Height := 13.626831, [1,8].Sample_FlowRate := 0.24634185, [1,8].Sample_FillTime := 66.0, [1,8].DisplacedCarbonVol := 43.64021, [1,8].DisplacedCarbonMass := 21.820105, [1,8].SampleDuration := 1065, [1,9].Run_ID := 2743, [1,9].Carbon_VOL_ml := 56.998867, [1,9].Carbon_MASS := 28.499434, [1,9].Carbon_DIST := 2.646463, [1,9].Hour := 12, [1,9].Min := 1, [1,9].Day := 21, [1,9].Month := 11, [1,9].Year := 2021, [1,9].Sample_DO := 5.8117228, [1,9].Sample_pH := 9.21795, [1,9].Sample_VOL := 10.768877, [1,9].Density := 312.91998, [1,9].EmptyDist := 1410.0, [1,9].FullDist := 1388.4265, [1,9].Carbon_mLperL := 5.292926, [1,9].Slurry_Weight := -10.52187, [1,9].Sample_Tank := 1, [1,9].Carbon_Height := 21.573486, [1,9].Sample_FlowRate := 0.053817473, [1,9].Sample_FillTime := 200.1, [1,9].DisplacedCarbonVol := 22.788153, [1,9].DisplacedCarbonMass := 11.394076, [1,9].SampleDuration := 972, [1,10].Run_ID := 2731, [1,10].Carbon_VOL_ml := 41.424404, [1,10].Carbon_MASS := 20.712202, [1,10].Carbon_DIST := 1.2368023, [1,10].Hour := 9, [1,10].Min := 1, [1,10].Day := 21, [1,10].Month := 11, [1,10].Year := 2021, [1,10].Sample_DO := 5.7468586, [1,10].Sample_pH := 9.315619, [1,10].Sample_VOL := 16.746574, [1,10].Density := 400.777, [1,10].EmptyDist := 1410.0, [1,10].FullDist := 1394.3213, [1,10].ErrorFlag := 1, [1,10].Carbon_mLperL := 2.4736047, [1,10].Slurry_Weight := -10.52187, [1,10].Sample_Tank := 1,
        [1,10].Carbon_Height := 15.678711, [1,10].Sample_FlowRate := 0.17098461, [1,10].Sample_FillTime := 97.942, [1,10].DisplacedCarbonVol := 33.83587, [1,10].DisplacedCarbonMass := 16.917934, [1,10].SampleDuration := 1077, [1,11].Run_ID := 2730, [1,11].Carbon_VOL_ml := 67.3756, [1,11].Carbon_MASS := 33.6878, [1,11].Carbon_DIST := 2.0996451, [1,11].Hour := 8, [1,11].Min := 45, [1,11].Day := 21, [1,11].Month := 11, [1,11].Year := 2021, [1,11].Sample_DO := 5.765432, [1,11].Sample_pH := 9.3252535, [1,11].Sample_VOL := 16.044521, [1,11].Density := 390.45862, [1,11].EmptyDist := 1410.0, [1,11].FullDist := 1384.499, [1,11].Carbon_mLperL := 4.1992903, [1,11].Slurry_Weight := -10.52187, [1,11].Sample_Tank := 1, [1,11].Carbon_Height := 25.500977, [1,11].Sample_FlowRate := 0.08000579, [1,11].Sample_FillTime := 200.542, [1,11].DisplacedCarbonVol := 26.877403, [1,11].DisplacedCarbonMass := 13.438702, [1,11].SampleDuration := 974, [1,12].Run_ID := 2721, [1,12].Carbon_VOL_ml := 11.860331, [1,12].Carbon_MASS := 5.9301653, [1,12].Carbon_DIST := 0.36512563, [1,12].Hour := 5, [1,12].Min := 39, [1,12].Day := 21, [1,12].Month := 11, [1,12].Year := 2021, [1,12].Sample_DO := 5.3639526, [1,12].Sample_pH := 9.215738, [1,12].Sample_VOL := 16.241438, [1,12].Density := 393.35278, [1,12].EmptyDist := 1410.0, [1,12].FullDist := 1405.511, [1,12].ErrorFlag := 1, [1,12].Carbon_mLperL := 0.73025125, [1,12].Slurry_Weight := -10.52187, [1,12].Sample_Tank := 1, [1,12].Carbon_Height := 4.4890137, [1,12].Sample_FlowRate := 0.23089246, [1,12].Sample_FillTime := 70.342, [1,12].DisplacedCarbonVol := 13.488761, [1,12].DisplacedCarbonMass := 6.7443805, [1,12].SampleDuration := 978, [1,13].Run_ID := 2720, [1,13].Carbon_VOL_ml := 47.871567, [1,13].Carbon_MASS := 23.935783, [1,13].Carbon_DIST := 1.4508041, [1,13].Hour := 5,
        [1,13].Min := 23, [1,13].Day := 21, [1,13].Month := 11, [1,13].Year := 2021, [1,13].Sample_DO := 5.5159597, [1,13].Sample_pH := 9.224604, [1,13].Sample_VOL := 16.498287, [1,13].Density := 397.1278, [1,13].EmptyDist := 1410.0, [1,13].FullDist := 1391.8811, [1,13].Carbon_mLperL := 2.9016082, [1,13].Slurry_Weight := -10.52187, [1,13].Sample_Tank := 1, [1,13].Carbon_Height := 18.118896, [1,13].Sample_FlowRate := 0.14745885, [1,13].Sample_FillTime := 111.884, [1,13].DisplacedCarbonVol := 34.229424, [1,13].DisplacedCarbonMass := 17.114712, [1,13].SampleDuration := 973, [1,14].Run_ID := 2710, [1,14].Carbon_VOL_ml := 247.05669, [1,14].Carbon_MASS := 123.52834, [1,14].Carbon_DIST := 7.0518622, [1,14].Hour := 2, [1,14].Min := 53, [1,14].Day := 21, [1,14].Month := 11, [1,14].Year := 2021, [1,14].Sample_DO := 6.247373, [1,14].Sample_pH := 9.337758, [1,14].Sample_VOL := 17.517124, [1,14].Density := 412.1021, [1,14].EmptyDist := 1410.0, [1,14].FullDist := 1316.4916, [1,14].ErrorFlag := 1, [1,14].Carbon_mLperL := 14.1037245, [1,14].Slurry_Weight := -10.52187, [1,14].Sample_Tank := 1, [1,14].Carbon_Height := 93.50842, [1,14].Sample_FlowRate := 2.3858788, [1,14].Sample_FillTime := 7.342001, [1,14].DisplacedCarbonVol := 2691.9822, [1,14].DisplacedCarbonMass := 1345.9911, [1,14].SampleDuration := 874, [1,15].Run_ID := 2709, [1,15].Carbon_VOL_ml := 221.10065, [1,15].Carbon_MASS := 110.55032, [1,15].Carbon_DIST := 6.3451, [1,15].Hour := 2, [1,15].Min := 38, [1,15].Day := 21, [1,15].Month := 11, [1,15].Year := 2021, [1,15].Sample_DO := 6.688827, [1,15].Sample_pH := 9.289061, [1,15].Sample_VOL := 17.422945, [1,15].Density := 410.71796, [1,15].EmptyDist := 1410.0, [1,15].FullDist := 1326.3157, [1,15].Carbon_mLperL := 12.6902,
        [1,15].Slurry_Weight := -10.52187, [1,15].Sample_Tank := 1, [1,15].Carbon_Height := 83.684326, [1,15].Sample_FlowRate := 2.5842395, [1,15].Sample_FillTime := 6.742001, [1,15].DisplacedCarbonVol := 2623.5613, [1,15].DisplacedCarbonMass := 1311.7806, [1,15].SampleDuration := 972, [1,16].Run_ID := 2697, [1,16].Hour := 23, [1,16].Min := 44, [1,16].Day := 20, [1,16].Month := 11, [1,16].Year := 2021, [1,16].Sample_DO := 5.8032174, [1,16].Sample_pH := 9.19808, [1,16].Sample_VOL := 16.575342, [1,16].Density := 398.26035, [1,16].EmptyDist := 1410.0, [1,16].FullDist := 1423.3958, [1,16].ErrorFlag := 1, [1,16].Slurry_Weight := -10.52187, [1,16].Sample_Tank := 1, [1,16].Carbon_Height := -13.395752, [1,16].Sample_FlowRate := 0.18665925, [1,16].Sample_FillTime := 88.8, [1,16].SampleDuration := 1011, [1,17].Run_ID := 2696, [1,17].Carbon_VOL_ml := 2.1460445, [1,17].Carbon_MASS := 1.0730222, [1,17].Carbon_DIST := 0.06592794, [1,17].Hour := 23, [1,17].Min := 28, [1,17].Day := 20, [1,17].Month := 11, [1,17].Year := 2021, [1,17].Sample_DO := 5.560534, [1,17].Sample_pH := 9.20327, [1,17].Sample_VOL := 16.275684, [1,17].Density := 393.8561, [1,17].EmptyDist := 1410.0, [1,17].FullDist := 1409.1877, [1,17].Carbon_mLperL := 0.13185588, [1,17].Slurry_Weight := -10.52187, [1,17].Sample_Tank := 1, [1,17].Carbon_Height := 0.81225586, [1,17].Sample_FlowRate := 0.11421533, [1,17].Sample_FillTime := 142.5, [1,17].DisplacedCarbonVol := 1.2047969, [1,17].DisplacedCarbonMass := 0.60239846, [1,17].SampleDuration := 973, [1,18].Run_ID := 2685, [1,18].Hour := 20, [1,18].Min := 46, [1,18].Day := 20, [1,18].Month := 11, [1,18].Year := 2021, [1,18].Sample_DO := 5.492019, [1,18].Sample_pH := 9.205111, [1,18].Sample_VOL := 16.001713,
        [1,18].Density := 389.8294, [1,18].EmptyDist := 1410.0, [1,18].FullDist := 1447.144, [1,18].ErrorFlag := 1, [1,18].Slurry_Weight := -10.52187, [1,18].Sample_Tank := 1, [1,18].Carbon_Height := -37.144043, [1,18].Sample_FlowRate := 0.11788328, [1,18].Sample_FillTime := 135.742, [1,18].SampleDuration := 1066, [1,19].Run_ID := 2684, [1,19].Carbon_VOL_ml := 28.820017, [1,19].Carbon_MASS := 14.410008, [1,19].Carbon_DIST := 0.9741219, [1,19].Hour := 20, [1,19].Min := 29, [1,19].Day := 20, [1,19].Month := 11, [1,19].Year := 2021, [1,19].Sample_DO := 5.460399, [1,19].Sample_pH := 9.207338, [1,19].Sample_VOL := 14.792818, [1,19].Density := 372.06174, [1,19].EmptyDist := 1410.0, [1,19].FullDist := 1399.0919, [1,19].Carbon_mLperL := 1.9482439, [1,19].Slurry_Weight := -10.52187, [1,19].Sample_Tank := 1, [1,19].Carbon_Height := 10.908081, [1,19].Sample_FlowRate := 0.07392713, [1,19].Sample_FillTime := 200.1, [1,19].DisplacedCarbonVol := 11.522246, [1,19].DisplacedCarbonMass := 5.761123, [1,19].SampleDuration := 972, [2,0].Run_ID := 2761, [2,0].Carbon_VOL_ml := 175.5638, [2,0].Carbon_MASS := 87.7819, [2,0].Carbon_DIST := 5.193985, [2,0].Hour := 16, [2,0].Min := 28, [2,0].Day := 21, [2,0].Month := 11, [2,0].Year := 2021, [2,0].Sample_DO := 6.1882257, [2,0].Sample_pH := 9.219038, [2,0].Sample_VOL := 16.900684, [2,0].Density := 403.04202, [2,0].EmptyDist := 1410.0, [2,0].FullDist := 1343.5509, [2,0].Carbon_mLperL := 10.38797, [2,0].Slurry_Weight := -10.52187, [2,0].Sample_Tank := 2, [2,0].Carbon_Height := 66.4491, [2,0].Sample_FlowRate := 1.8778536, [2,0].Sample_FillTime := 9.000001, [2,0].DisplacedCarbonVol := 1560.5671, [2,0].DisplacedCarbonMass := 780.28357, [2,0].SampleDuration := 934, [2,1].Run_ID := 2746, [2,1].Carbon_VOL_ml := 253.23488,
        [2,1].Carbon_MASS := 126.61744, [2,1].Carbon_DIST := 7.450336, [2,1].Hour := 12, [2,1].Min := 46, [2,1].Day := 21, [2,1].Month := 11, [2,1].Year := 2021, [2,1].Sample_DO := 6.166438, [2,1].Sample_pH := 9.177105, [2,1].Sample_VOL := 16.994864, [2,1].Density := 404.42624, [2,1].EmptyDist := 1410.0, [2,1].FullDist := 1314.1532, [2,1].ErrorFlag := 1, [2,1].Carbon_mLperL := 14.900672, [2,1].Slurry_Weight := -10.52187, [2,1].Sample_Tank := 2, [2,1].Carbon_Height := 95.8468, [2,1].Sample_FlowRate := 1.4331981, [2,1].Sample_FillTime := 11.858001, [2,1].DisplacedCarbonVol := 1708.4491, [2,1].DisplacedCarbonMass := 854.22455, [2,1].SampleDuration := 875, [2,2].Run_ID := 2745, [2,2].Carbon_VOL_ml := 216.11836, [2,2].Carbon_MASS := 108.05918, [2,2].Carbon_DIST := 6.2419944, [2,2].Hour := 12, [2,2].Min := 31, [2,2].Day := 21, [2,2].Month := 11, [2,2].Year := 2021, [2,2].Sample_DO := 6.544005, [2,2].Sample_pH := 9.146523, [2,2].Sample_VOL := 17.311644, [2,2].Density := 409.0821, [2,2].EmptyDist := 1410.0, [2,2].FullDist := 1328.2014, [2,2].Carbon_mLperL := 12.483989, [2,2].Slurry_Weight := -10.52187, [2,2].Sample_Tank := 2, [2,2].Carbon_Height := 81.798584, [2,2].Sample_FlowRate := 1.4796276, [2,2].Sample_FillTime := 11.700001, [2,2].DisplacedCarbonVol := 1477.7324, [2,2].DisplacedCarbonMass := 738.8662, [2,2].SampleDuration := 933, [2,3].Run_ID := 2732, [2,3].Carbon_VOL_ml := 116.71398, [2,3].Carbon_MASS := 58.35699, [2,3].Carbon_DIST := 3.3643122, [2,3].Hour := 9, [2,3].Min := 16, [2,3].Day := 21, [2,3].Month := 11, [2,3].Year := 2021, [2,3].Sample_DO := 5.9324217, [2,3].Sample_pH := 9.155974, [2,3].Sample_VOL := 17.34589, [2,3].Density := 409.58542,
        [2,3].EmptyDist := 1410.0, [2,3].FullDist := 1365.825, [2,3].Carbon_mLperL := 6.7286243, [2,3].Slurry_Weight := -10.52187, [2,3].Sample_Tank := 2, [2,3].Carbon_Height := 44.17505, [2,3].Sample_FlowRate := 1.3766578, [2,3].Sample_FillTime := 12.600001, [2,3].DisplacedCarbonVol := 741.0411, [2,3].DisplacedCarbonMass := 370.52054, [2,3].SampleDuration := 970, [2,4].Run_ID := 2722, [2,4].Carbon_VOL_ml := 217.00594, [2,4].Carbon_MASS := 108.50297, [2,4].Carbon_DIST := 6.252169, [2,4].Hour := 5, [2,4].Min := 53, [2,4].Day := 21, [2,4].Month := 11, [2,4].Year := 2021, [2,4].Sample_DO := 5.9623084, [2,4].Sample_pH := 9.266289, [2,4].Sample_VOL := 17.354452, [2,4].Density := 409.71127, [2,4].EmptyDist := 1410.0, [2,4].FullDist := 1327.8655, [2,4].Carbon_mLperL := 12.504338, [2,4].Slurry_Weight := -10.52187, [2,4].Sample_Tank := 2, [2,4].Carbon_Height := 82.13452, [2,4].Sample_FlowRate := 1.8983209, [2,4].Sample_FillTime := 9.142001, [2,4].DisplacedCarbonVol := 1898.9797, [2,4].DisplacedCarbonMass := 949.48987, [2,4].SampleDuration := 936, [2,5].Run_ID := 2711, [2,5].Carbon_VOL_ml := 391.68314, [2,5].Carbon_MASS := 195.84157, [2,5].Carbon_DIST := 11.340752, [2,5].Hour := 3, [2,5].Min := 7, [2,5].Day := 21, [2,5].Month := 11, [2,5].Year := 2021, [2,5].Sample_DO := 6.859827, [2,5].Sample_pH := 9.31351, [2,5].Sample_VOL := 17.268835, [2,5].Density := 408.45288, [2,5].EmptyDist := 1410.0, [2,5].FullDist := 1261.752, [2,5].Carbon_mLperL := 22.681503, [2,5].Slurry_Weight := -10.52187, [2,5].Sample_Tank := 2, [2,5].Carbon_Height := 148.24805, [2,5].Sample_FlowRate := 2.1319547, [2,5].Sample_FillTime := 8.100001, [2,5].DisplacedCarbonVol := 3868.475, [2,5].DisplacedCarbonMass := 1934.2375, [2,5].SampleDuration := 886, [2,6].Run_ID := 2699,
        [2,6].Carbon_VOL_ml := 343.06137, [2,6].Carbon_MASS := 171.53069, [2,6].Carbon_DIST := 9.825789, [2,6].Min := 13, [2,6].Day := 21, [2,6].Month := 11, [2,6].Year := 2021, [2,6].Sample_DO := 6.523859, [2,6].Sample_pH := 9.111001, [2,6].Sample_VOL := 17.457191, [2,6].Density := 411.22125, [2,6].EmptyDist := 1410.0, [2,6].FullDist := 1280.1548, [2,6].ErrorFlag := 1, [2,6].Carbon_mLperL := 19.651579, [2,6].Slurry_Weight := -10.52187, [2,6].Sample_Tank := 2, [2,6].Carbon_Height := 129.84521, [2,6].Sample_FlowRate := 1.5124927, [2,6].Sample_FillTime := 11.542001, [2,6].DisplacedCarbonVol := 2377.8296, [2,6].DisplacedCarbonMass := 1188.9148, [2,6].SampleDuration := 878, [2,7].Run_ID := 2698, [2,7].Carbon_VOL_ml := 280.90802, [2,7].Carbon_MASS := 140.45401, [2,7].Carbon_DIST := 8.227196, [2,7].Hour := 23, [2,7].Min := 58, [2,7].Day := 20, [2,7].Month := 11, [2,7].Year := 2021, [2,7].Sample_DO := 6.320257, [2,7].Sample_pH := 9.133423, [2,7].Sample_VOL := 17.071918, [2,7].Density := 405.55872, [2,7].EmptyDist := 1410.0, [2,7].FullDist := 1303.6792, [2,7].Carbon_mLperL := 16.454391, [2,7].Slurry_Weight := -10.52187, [2,7].Sample_Tank := 2, [2,7].Carbon_Height := 106.3208, [2,7].Sample_FlowRate := 1.4396962, [2,7].Sample_FillTime := 11.858001, [2,7].DisplacedCarbonVol := 1895.146, [2,7].DisplacedCarbonMass := 947.573, [2,7].SampleDuration := 964, [2,8].Run_ID := 2686, [2,8].Carbon_VOL_ml := 129.15356, [2,8].Carbon_MASS := 64.57678, [2,8].Carbon_DIST := 3.6721363, [2,8].Hour := 21, [2,8].Day := 20, [2,8].Month := 11, [2,8].Year := 2021, [2,8].Sample_DO := 8.327417, [2,8].Sample_pH := 9.21543, [2,8].Sample_VOL := 17.585617, [2,8].Density := 413.10876, [2,8].EmptyDist := 1410.0,
        [2,8].FullDist := 1361.1167, [2,8].Carbon_mLperL := 7.3442726, [2,8].Slurry_Weight := -10.52187, [2,8].Sample_Tank := 2, [2,8].Carbon_Height := 48.8833, [2,8].Sample_FlowRate := 1.805134, [2,8].Sample_FillTime := 9.742001, [2,8].DisplacedCarbonVol := 1060.5918, [2,8].DisplacedCarbonMass := 530.2959, [2,8].SampleDuration := 1003, [2,9].Run_ID := 2674, [2,9].Carbon_VOL_ml := 139.23296, [2,9].Carbon_MASS := 69.61648, [2,9].Carbon_DIST := 4.100456, [2,9].Hour := 17, [2,9].Min := 56, [2,9].Day := 20, [2,9].Month := 11, [2,9].Year := 2021, [2,9].Sample_DO := 7.2013807, [2,9].Sample_pH := 9.284256, [2,9].Sample_VOL := 16.97774, [2,9].Density := 404.17456, [2,9].EmptyDist := 1410.0, [2,9].FullDist := 1357.3018, [2,9].ErrorFlag := 1, [2,9].Carbon_mLperL := 8.200912, [2,9].Slurry_Weight := -10.52187, [2,9].Sample_Tank := 2, [2,9].Carbon_Height := 52.698242, [2,9].Sample_FlowRate := 2.2216353, [2,9].Sample_FillTime := 7.642001, [2,9].DisplacedCarbonVol := 1457.5549, [2,9].DisplacedCarbonMass := 728.77747, [2,9].SampleDuration := 870, [2,10].Run_ID := 2673, [2,10].Carbon_VOL_ml := 179.65495, [2,10].Carbon_MASS := 89.82748, [2,10].Carbon_DIST := 5.2485485, [2,10].Hour := 17, [2,10].Min := 41, [2,10].Day := 20, [2,10].Month := 11, [2,10].Year := 2021, [2,10].Sample_DO := 7.3462377, [2,10].Sample_pH := 9.272914, [2,10].Sample_VOL := 17.114727, [2,10].Density := 406.18787, [2,10].EmptyDist := 1410.0, [2,10].FullDist := 1342.0024, [2,10].Carbon_mLperL := 10.497097, [2,10].Slurry_Weight := -10.52187, [2,10].Sample_Tank := 2, [2,10].Carbon_Height := 67.99756, [2,10].Sample_FlowRate := 2.1941955, [2,10].Sample_FillTime := 7.800001, [2,10].DisplacedCarbonVol := 1842.6147, [2,10].DisplacedCarbonMass := 921.3074, [2,10].SampleDuration := 875, [2,11].Run_ID := 2661,
        [2,11].Carbon_VOL_ml := 364.40445, [2,11].Carbon_MASS := 182.20222, [2,11].Carbon_DIST := 10.737246, [2,11].Hour := 14, [2,11].Min := 46, [2,11].Day := 20, [2,11].Month := 11, [2,11].Year := 2021, [2,11].Sample_DO := 5.1347313, [2,11].Sample_pH := 9.260895, [2,11].Sample_VOL := 16.969177, [2,11].Density := 404.04868, [2,11].EmptyDist := 1410.0, [2,11].FullDist := 1272.0767, [2,11].ErrorFlag := 1, [2,11].Carbon_mLperL := 21.474491, [2,11].Slurry_Weight := -10.52187, [2,11].Sample_Tank := 2, [2,11].Carbon_Height := 137.92334, [2,11].Sample_FlowRate := 1.95048, [2,11].Sample_FillTime := 8.700001, [2,11].DisplacedCarbonVol := 3350.8455, [2,11].DisplacedCarbonMass := 1675.4227, [2,11].SampleDuration := 874, [2,12].Run_ID := 2660, [2,12].Hour := 14, [2,12].Min := 31, [2,12].Day := 20, [2,12].Month := 11, [2,12].Year := 2021, [2,12].Sample_DO := 5.443984, [2,12].Sample_pH := 9.228107, [2,12].Sample_VOL := 17.28596, [2,12].Density := 408.70456, [2,12].EmptyDist := 1410.0, [2,12].FullDist := 1411.1375, [2,12].Slurry_Weight := -10.52187, [2,12].Sample_Tank := 2, [2,12].Carbon_Height := -1.1374512, [2,12].Sample_FlowRate := 1.9514515, [2,12].Sample_FillTime := 8.858001, [2,12].SampleDuration := 872, [2,13].Run_ID := 2649, [2,13].Carbon_VOL_ml := 248.44545, [2,13].Carbon_MASS := 124.222725, [2,13].Carbon_DIST := 7.01267, [2,13].Hour := 11, [2,13].Min := 45, [2,13].Day := 20, [2,13].Month := 11, [2,13].Year := 2021, [2,13].Sample_DO := 5.730744, [2,13].Sample_pH := 9.090882, [2,13].Sample_VOL := 17.71404, [2,13].Density := 414.99634, [2,13].EmptyDist := 1410.0, [2,13].FullDist := 1315.966, [2,13].Carbon_mLperL := 14.02534, [2,13].Slurry_Weight := -10.52187, [2,13].Sample_Tank := 2,
        [2,13].Carbon_Height := 94.03406, [2,13].Sample_FlowRate := 1.2836261, [2,13].Sample_FillTime := 13.800001, [2,13].DisplacedCarbonVol := 1440.2634, [2,13].DisplacedCarbonMass := 720.1317, [2,13].SampleDuration := 977, [2,14].Run_ID := 2639, [2,14].Carbon_VOL_ml := 319.21204, [2,14].Carbon_MASS := 159.60602, [2,14].Carbon_DIST := 8.966803, [2,14].Hour := 9, [2,14].Min := 12, [2,14].Day := 20, [2,14].Month := 11, [2,14].Year := 2021, [2,14].Sample_DO := 5.754249, [2,14].Sample_pH := 9.144333, [2,14].Sample_VOL := 17.799658, [2,14].Density := 416.2546, [2,14].EmptyDist := 1410.0, [2,14].FullDist := 1289.1815, [2,14].Carbon_mLperL := 17.933605, [2,14].Slurry_Weight := -10.52187, [2,14].Sample_Tank := 2, [2,14].Carbon_Height := 120.81848, [2,14].Sample_FlowRate := 1.1633762, [2,14].Sample_FillTime := 15.300001, [2,14].DisplacedCarbonVol := 1669.0824, [2,14].DisplacedCarbonMass := 834.5412, [2,14].SampleDuration := 1015, [2,15].Run_ID := 2629, [2,15].Carbon_VOL_ml := 307.0295, [2,15].Carbon_MASS := 153.51476, [2,15].Carbon_DIST := 8.716832, [2,15].Hour := 6, [2,15].Min := 8, [2,15].Day := 20, [2,15].Month := 11, [2,15].Year := 2021, [2,15].Sample_DO := 5.819656, [2,15].Sample_pH := 9.193593, [2,15].Sample_VOL := 17.611301, [2,15].Density := 413.4863, [2,15].EmptyDist := 1410.0, [2,15].FullDist := 1293.7925, [2,15].Carbon_mLperL := 17.433664, [2,15].Slurry_Weight := -10.52187, [2,15].Sample_Tank := 2, [2,15].Carbon_Height := 116.20752, [2,15].Sample_FlowRate := 1.2761811, [2,15].Sample_FillTime := 13.800001, [2,15].DisplacedCarbonVol := 1779.8811, [2,15].DisplacedCarbonMass := 889.94055, [2,15].SampleDuration := 937, [2,16].Run_ID := 2620, [2,16].Carbon_VOL_ml := 221.25609, [2,16].Carbon_MASS := 110.628044, [2,16].Carbon_DIST := 6.2938895, [2,16].Hour := 3, [2,16].Min := 53,
